(* Logix 5000 project; controller QW361 vendor 1 type 14 code 107 rev 32.11; software revision 32.00; part 18 of 20 *)

        [136].log_data[5].minminute := 7, [136].log_data[5].valid := 1, [136].log_data[6].valid := 1, [136].log_data[7].valid := 1, [136].log_data[8].valid := 1, [136].log_data[9].valid := 1, [136].log_data[10].valid := 1, [136].log_data[11].valid := 1, [136].log_data[12].valid := 1, [136].log_data[13].valid := 1, [136].log_data[14].valid := 1, [136].log_data[15].valid := 1, [136].log_data[16].valid := 1, [136].log_data[17].valid := 1, [136].log_data[18].valid := 1, [136].log_data[19].valid := 1, [136].time.Year := 2022, [136].time.Month := 5, [136].time.Day := 2, [136].time.Hour := 9, [136].time.Minute := 59, [136].time.Second := 59, [136].time.DST_ON := 1, [137].log_data[0].min := 1.0, [137].log_data[0].max := 1.0, [137].log_data[0].total := 3599.999, [137].log_data[0].time := 3599.999, [137].log_data[0].valid := 1, [137].log_data[1].max := 1.0, [137].log_data[1].total := 500.5, [137].log_data[1].time := 3599.999, [137].log_data[1].maxminute := 16, [137].log_data[1].valid := 1, [137].log_data[2].time := 3599.999, [137].log_data[2].valid := 1, [137].log_data[3].time := 3599.999, [137].log_data[3].valid := 1, [137].log_data[4].min := 0.48812497, [137].log_data[4].max := 1.0081251, [137].log_data[4].total := 2728.107, [137].log_data[4].time := 3599.999, [137].log_data[4].minminute := 25, [137].log_data[4].maxminute := 16, [137].log_data[4].valid := 1, [137].log_data[5].max := 7.1587505, [137].log_data[5].total := 3522.9197, [137].log_data[5].time := 3599.999, [137].log_data[5].maxminute := 17, [137].log_data[5].valid := 1, [137].log_data[6].valid := 1, [137].log_data[7].valid := 1, [137].log_data[8].valid := 1, [137].log_data[9].valid := 1, [137].log_data[10].valid := 1, [137].log_data[11].valid := 1, [137].log_data[12].valid := 1, [137].log_data[13].valid := 1, [137].log_data[14].valid := 1, [137].log_data[15].valid := 1, [137].log_data[16].valid := 1,
        [137].log_data[17].valid := 1, [137].log_data[18].valid := 1, [137].log_data[19].valid := 1, [137].time.Year := 2022, [137].time.Month := 5, [137].time.Day := 2, [137].time.Hour := 10, [137].time.Minute := 59, [137].time.Second := 59, [137].time.DST_ON := 1, [138].log_data[0].min := 1.0, [138].log_data[0].max := 1.0, [138].log_data[0].total := 3599.999, [138].log_data[0].time := 3599.999, [138].log_data[0].valid := 1, [138].log_data[1].time := 3599.999, [138].log_data[1].valid := 1, [138].log_data[2].max := 1.0, [138].log_data[2].total := 495.0, [138].log_data[2].time := 3599.999, [138].log_data[2].maxminute := 43, [138].log_data[2].valid := 1, [138].log_data[3].time := 3599.999, [138].log_data[3].valid := 1, [138].log_data[4].min := 0.48749998, [138].log_data[4].max := 1.0068749, [138].log_data[4].total := 3053.5842, [138].log_data[4].time := 3599.999, [138].log_data[4].minminute := 52, [138].log_data[4].maxminute := 43, [138].log_data[4].valid := 1, [138].log_data[5].max := 7.26375, [138].log_data[5].total := 3527.154, [138].log_data[5].time := 3599.999, [138].log_data[5].maxminute := 43, [138].log_data[5].valid := 1, [138].log_data[6].valid := 1, [138].log_data[7].valid := 1, [138].log_data[8].valid := 1, [138].log_data[9].valid := 1, [138].log_data[10].valid := 1, [138].log_data[11].valid := 1, [138].log_data[12].valid := 1, [138].log_data[13].valid := 1, [138].log_data[14].valid := 1, [138].log_data[15].valid := 1, [138].log_data[16].valid := 1, [138].log_data[17].valid := 1, [138].log_data[18].valid := 1, [138].log_data[19].valid := 1, [138].time.Year := 2022, [138].time.Month := 5, [138].time.Day := 2, [138].time.Hour := 11, [138].time.Minute := 59, [138].time.Second := 59, [138].time.DST_ON := 1, [139].log_data[0].min := 1.0, [139].log_data[0].max := 1.0, [139].log_data[0].total := 3599.999,
        [139].log_data[0].time := 3599.999, [139].log_data[0].valid := 1, [139].log_data[1].time := 3599.999, [139].log_data[1].valid := 1, [139].log_data[2].time := 3599.999, [139].log_data[2].valid := 1, [139].log_data[3].time := 3599.999, [139].log_data[3].valid := 1, [139].log_data[4].min := 0.56437504, [139].log_data[4].max := 0.9650001, [139].log_data[4].total := 2955.463, [139].log_data[4].time := 3599.999, [139].log_data[4].maxminute := 58, [139].log_data[4].valid := 1, [139].log_data[5].max := 0.0012500001, [139].log_data[5].total := 0.057499956, [139].log_data[5].time := 3599.999, [139].log_data[5].maxminute := 1, [139].log_data[5].valid := 1, [139].log_data[6].valid := 1, [139].log_data[7].valid := 1, [139].log_data[8].valid := 1, [139].log_data[9].valid := 1, [139].log_data[10].valid := 1, [139].log_data[11].valid := 1, [139].log_data[12].valid := 1, [139].log_data[13].valid := 1, [139].log_data[14].valid := 1, [139].log_data[15].valid := 1, [139].log_data[16].valid := 1, [139].log_data[17].valid := 1, [139].log_data[18].valid := 1, [139].log_data[19].valid := 1, [139].time.Year := 2022, [139].time.Month := 5, [139].time.Day := 2, [139].time.Hour := 12, [139].time.Minute := 59, [139].time.Second := 59, [139].time.DST_ON := 1, [140].log_data[0].min := 1.0, [140].log_data[0].max := 1.0, [140].log_data[0].total := 3600.0, [140].log_data[0].time := 3600.0, [140].log_data[0].valid := 1, [140].log_data[1].max := 1.0, [140].log_data[1].total := 501.0, [140].log_data[1].time := 3600.0, [140].log_data[1].maxminute := 9, [140].log_data[1].valid := 1, [140].log_data[2].time := 3600.0, [140].log_data[2].valid := 1, [140].log_data[3].time := 3600.0, [140].log_data[3].valid := 1, [140].log_data[4].min := 0.48749998, [140].log_data[4].max := 1.00875, [140].log_data[4].total := 2592.416, [140].log_data[4].time := 3600.0, [140].log_data[4].minminute := 18, [140].log_data[4].maxminute := 9,
        [140].log_data[4].valid := 1, [140].log_data[5].max := 7.1550007, [140].log_data[5].total := 3519.3843, [140].log_data[5].time := 3600.0, [140].log_data[5].maxminute := 10, [140].log_data[5].valid := 1, [140].log_data[6].valid := 1, [140].log_data[7].valid := 1, [140].log_data[8].valid := 1, [140].log_data[9].valid := 1, [140].log_data[10].valid := 1, [140].log_data[11].valid := 1, [140].log_data[12].valid := 1, [140].log_data[13].valid := 1, [140].log_data[14].valid := 1, [140].log_data[15].valid := 1, [140].log_data[16].valid := 1, [140].log_data[17].valid := 1, [140].log_data[18].valid := 1, [140].log_data[19].valid := 1, [140].time.Year := 2022, [140].time.Month := 5, [140].time.Day := 2, [140].time.Hour := 13, [140].time.Minute := 59, [140].time.Second := 59, [140].time.DST_ON := 1, [141].log_data[0].min := 1.0, [141].log_data[0].max := 1.0, [141].log_data[0].total := 3600.001, [141].log_data[0].time := 3600.001, [141].log_data[0].valid := 1, [141].log_data[1].time := 3600.001, [141].log_data[1].valid := 1, [141].log_data[2].time := 3600.001, [141].log_data[2].valid := 1, [141].log_data[3].time := 3600.001, [141].log_data[3].valid := 1, [141].log_data[4].min := 0.77937496, [141].log_data[4].max := 0.94875, [141].log_data[4].total := 3176.0435, [141].log_data[4].time := 3600.001, [141].log_data[4].maxminute := 56, [141].log_data[4].valid := 1, [141].log_data[5].max := 0.0012500001, [141].log_data[5].total := 0.14781292, [141].log_data[5].time := 3600.001, [141].log_data[5].valid := 1, [141].log_data[6].valid := 1, [141].log_data[7].valid := 1, [141].log_data[8].valid := 1, [141].log_data[9].valid := 1, [141].log_data[10].valid := 1, [141].log_data[11].valid := 1, [141].log_data[12].valid := 1, [141].log_data[13].valid := 1, [141].log_data[14].valid := 1, [141].log_data[15].valid := 1, [141].log_data[16].valid := 1, [141].log_data[17].valid := 1,
        [141].log_data[18].valid := 1, [141].log_data[19].valid := 1, [141].time.Year := 2022, [141].time.Month := 5, [141].time.Day := 2, [141].time.Hour := 14, [141].time.Minute := 59, [141].time.Second := 59, [141].time.DST_ON := 1, [142].log_data[0].min := 1.0, [142].log_data[0].max := 1.0, [142].log_data[0].total := 3600.0, [142].log_data[0].time := 3600.0, [142].log_data[0].valid := 1, [142].log_data[1].time := 3600.0, [142].log_data[1].valid := 1, [142].log_data[2].max := 1.0, [142].log_data[2].total := 480.0, [142].log_data[2].time := 3600.0, [142].log_data[2].maxminute := 26, [142].log_data[2].valid := 1, [142].log_data[3].time := 3600.0, [142].log_data[3].valid := 1, [142].log_data[4].min := 0.48749998, [142].log_data[4].max := 1.00625, [142].log_data[4].total := 2781.7415, [142].log_data[4].time := 3600.0, [142].log_data[4].minminute := 34, [142].log_data[4].maxminute := 26, [142].log_data[4].valid := 1, [142].log_data[5].max := 7.3075004, [142].log_data[5].total := 3444.1716, [142].log_data[5].time := 3600.0, [142].log_data[5].maxminute := 27, [142].log_data[5].valid := 1, [142].log_data[6].valid := 1, [142].log_data[7].valid := 1, [142].log_data[8].valid := 1, [142].log_data[9].valid := 1, [142].log_data[10].valid := 1, [142].log_data[11].valid := 1, [142].log_data[12].valid := 1, [142].log_data[13].valid := 1, [142].log_data[14].valid := 1, [142].log_data[15].valid := 1, [142].log_data[16].valid := 1, [142].log_data[17].valid := 1, [142].log_data[18].valid := 1, [142].log_data[19].valid := 1, [142].time.Year := 2022, [142].time.Month := 5, [142].time.Day := 2, [142].time.Hour := 15, [142].time.Minute := 59, [142].time.Second := 59, [142].time.DST_ON := 1, [143].log_data[0].min := 1.0, [143].log_data[0].max := 1.0, [143].log_data[0].total := 3599.999, [143].log_data[0].time := 3599.999,
        [143].log_data[0].valid := 1, [143].log_data[1].time := 3599.999, [143].log_data[1].valid := 1, [143].log_data[2].time := 3599.999, [143].log_data[2].valid := 1, [143].log_data[3].time := 3599.999, [143].log_data[3].valid := 1, [143].log_data[4].min := 0.64125, [143].log_data[4].max := 0.97937495, [143].log_data[4].total := 2973.9944, [143].log_data[4].time := 3599.999, [143].log_data[4].maxminute := 57, [143].log_data[4].valid := 1, [143].log_data[5].time := 3599.999, [143].log_data[5].valid := 1, [143].log_data[6].valid := 1, [143].log_data[7].valid := 1, [143].log_data[8].valid := 1, [143].log_data[9].valid := 1, [143].log_data[10].valid := 1, [143].log_data[11].valid := 1, [143].log_data[12].valid := 1, [143].log_data[13].valid := 1, [143].log_data[14].valid := 1, [143].log_data[15].valid := 1, [143].log_data[16].valid := 1, [143].log_data[17].valid := 1, [143].log_data[18].valid := 1, [143].log_data[19].valid := 1, [143].time.Year := 2022, [143].time.Month := 5, [143].time.Day := 2, [143].time.Hour := 16, [143].time.Minute := 59, [143].time.Second := 59, [143].time.DST_ON := 1, [144].log_data[0].min := 1.0, [144].log_data[0].max := 1.0, [144].log_data[0].total := 3600.0, [144].log_data[0].time := 3600.0, [144].log_data[0].valid := 1, [144].log_data[1].max := 1.0, [144].log_data[1].total := 497.5, [144].log_data[1].time := 3600.0, [144].log_data[1].maxminute := 6, [144].log_data[1].valid := 1, [144].log_data[2].time := 3600.0, [144].log_data[2].valid := 1, [144].log_data[3].time := 3600.0, [144].log_data[3].valid := 1, [144].log_data[4].min := 0.48749998, [144].log_data[4].max := 1.00875, [144].log_data[4].total := 2580.9526, [144].log_data[4].time := 3600.0, [144].log_data[4].minminute := 15, [144].log_data[4].maxminute := 6, [144].log_data[4].valid := 1, [144].log_data[5].max := 7.1587505, [144].log_data[5].total := 3498.0137, [144].log_data[5].time := 3600.0,
        [144].log_data[5].maxminute := 8, [144].log_data[5].valid := 1, [144].log_data[6].valid := 1, [144].log_data[7].valid := 1, [144].log_data[8].valid := 1, [144].log_data[9].valid := 1, [144].log_data[10].valid := 1, [144].log_data[11].valid := 1, [144].log_data[12].valid := 1, [144].log_data[13].valid := 1, [144].log_data[14].valid := 1, [144].log_data[15].valid := 1, [144].log_data[16].valid := 1, [144].log_data[17].valid := 1, [144].log_data[18].valid := 1, [144].log_data[19].valid := 1, [144].time.Year := 2022, [144].time.Month := 5, [144].time.Day := 2, [144].time.Hour := 17, [144].time.Minute := 59, [144].time.Second := 59, [144].time.DST_ON := 1, [145].log_data[0].min := 1.0, [145].log_data[0].max := 1.0, [145].log_data[0].total := 3600.0, [145].log_data[0].time := 3600.0, [145].log_data[0].valid := 1, [145].log_data[1].time := 3600.0, [145].log_data[1].valid := 1, [145].log_data[2].max := 1.0, [145].log_data[2].total := 489.5, [145].log_data[2].time := 3600.0, [145].log_data[2].maxminute := 45, [145].log_data[2].valid := 1, [145].log_data[3].time := 3600.0, [145].log_data[3].valid := 1, [145].log_data[4].min := 0.48749998, [145].log_data[4].max := 1.00875, [145].log_data[4].total := 3124.9949, [145].log_data[4].time := 3600.0, [145].log_data[4].minminute := 53, [145].log_data[4].maxminute := 45, [145].log_data[4].valid := 1, [145].log_data[5].max := 7.2675, [145].log_data[5].total := 3485.3735, [145].log_data[5].time := 3600.0, [145].log_data[5].maxminute := 46, [145].log_data[5].valid := 1, [145].log_data[6].valid := 1, [145].log_data[7].valid := 1, [145].log_data[8].valid := 1, [145].log_data[9].valid := 1, [145].log_data[10].valid := 1, [145].log_data[11].valid := 1, [145].log_data[12].valid := 1, [145].log_data[13].valid := 1, [145].log_data[14].valid := 1, [145].log_data[15].valid := 1, [145].log_data[16].valid := 1,
        [145].log_data[17].valid := 1, [145].log_data[18].valid := 1, [145].log_data[19].valid := 1, [145].time.Year := 2022, [145].time.Month := 5, [145].time.Day := 2, [145].time.Hour := 18, [145].time.Minute := 59, [145].time.Second := 59, [145].time.DST_ON := 1, [146].log_data[0].min := 1.0, [146].log_data[0].max := 1.0, [146].log_data[0].total := 3600.0, [146].log_data[0].time := 3600.0, [146].log_data[0].valid := 1, [146].log_data[1].time := 3600.0, [146].log_data[1].valid := 1, [146].log_data[2].time := 3600.0, [146].log_data[2].valid := 1, [146].log_data[3].time := 3600.0, [146].log_data[3].valid := 1, [146].log_data[4].min := 0.53374994, [146].log_data[4].max := 0.933125, [146].log_data[4].total := 2734.3828, [146].log_data[4].time := 3600.0, [146].log_data[4].maxminute := 58, [146].log_data[4].valid := 1, [146].log_data[5].time := 3600.0, [146].log_data[5].valid := 1, [146].log_data[6].valid := 1, [146].log_data[7].valid := 1, [146].log_data[8].valid := 1, [146].log_data[9].valid := 1, [146].log_data[10].valid := 1, [146].log_data[11].valid := 1, [146].log_data[12].valid := 1, [146].log_data[13].valid := 1, [146].log_data[14].valid := 1, [146].log_data[15].valid := 1, [146].log_data[16].valid := 1, [146].log_data[17].valid := 1, [146].log_data[18].valid := 1, [146].log_data[19].valid := 1, [146].time.Year := 2022, [146].time.Month := 5, [146].time.Day := 2, [146].time.Hour := 19, [146].time.Minute := 59, [146].time.Second := 59, [146].time.DST_ON := 1, [147].log_data[0].min := 1.0, [147].log_data[0].max := 1.0, [147].log_data[0].total := 3600.0, [147].log_data[0].time := 3600.0, [147].log_data[0].valid := 1, [147].log_data[1].max := 1.0, [147].log_data[1].total := 512.0, [147].log_data[1].time := 3600.0, [147].log_data[1].maxminute := 17, [147].log_data[1].valid := 1,
        [147].log_data[2].time := 3600.0, [147].log_data[2].valid := 1, [147].log_data[3].time := 3600.0, [147].log_data[3].valid := 1, [147].log_data[4].min := 0.48749998, [147].log_data[4].max := 1.00875, [147].log_data[4].total := 2863.854, [147].log_data[4].time := 3600.0, [147].log_data[4].minminute := 26, [147].log_data[4].maxminute := 18, [147].log_data[4].valid := 1, [147].log_data[5].max := 7.1587505, [147].log_data[5].total := 3600.5417, [147].log_data[5].time := 3600.0, [147].log_data[5].maxminute := 18, [147].log_data[5].valid := 1, [147].log_data[6].valid := 1, [147].log_data[7].valid := 1, [147].log_data[8].valid := 1, [147].log_data[9].valid := 1, [147].log_data[10].valid := 1, [147].log_data[11].valid := 1, [147].log_data[12].valid := 1, [147].log_data[13].valid := 1, [147].log_data[14].valid := 1, [147].log_data[15].valid := 1, [147].log_data[16].valid := 1, [147].log_data[17].valid := 1, [147].log_data[18].valid := 1, [147].log_data[19].valid := 1, [147].time.Year := 2022, [147].time.Month := 5, [147].time.Day := 2, [147].time.Hour := 20, [147].time.Minute := 59, [147].time.Second := 59, [147].time.DST_ON := 1, [148].log_data[0].min := 1.0, [148].log_data[0].max := 1.0, [148].log_data[0].total := 3600.0, [148].log_data[0].time := 3600.0, [148].log_data[0].valid := 1, [148].log_data[1].time := 3600.0, [148].log_data[1].valid := 1, [148].log_data[2].max := 1.0, [148].log_data[2].total := 498.0, [148].log_data[2].time := 3600.0, [148].log_data[2].maxminute := 20, [148].log_data[2].valid := 1, [148].log_data[3].time := 3600.0, [148].log_data[3].valid := 1, [148].log_data[4].min := 0.48749998, [148].log_data[4].max := 1.00875, [148].log_data[4].total := 2776.5615, [148].log_data[4].time := 3600.0, [148].log_data[4].minminute := 28, [148].log_data[4].maxminute := 20, [148].log_data[4].valid := 1, [148].log_data[5].max := 7.2425003, [148].log_data[5].total := 3543.449,
        [148].log_data[5].time := 3600.0, [148].log_data[5].maxminute := 21, [148].log_data[5].valid := 1, [148].log_data[6].valid := 1, [148].log_data[7].valid := 1, [148].log_data[8].valid := 1, [148].log_data[9].valid := 1, [148].log_data[10].valid := 1, [148].log_data[11].valid := 1, [148].log_data[12].valid := 1, [148].log_data[13].valid := 1, [148].log_data[14].valid := 1, [148].log_data[15].valid := 1, [148].log_data[16].valid := 1, [148].log_data[17].valid := 1, [148].log_data[18].valid := 1, [148].log_data[19].valid := 1, [148].time.Year := 2022, [148].time.Month := 5, [148].time.Day := 2, [148].time.Hour := 21, [148].time.Minute := 59, [148].time.Second := 59, [148].time.DST_ON := 1, [149].log_data[0].min := 1.0, [149].log_data[0].max := 1.0, [149].log_data[0].total := 3600.0, [149].log_data[0].time := 3600.0, [149].log_data[0].valid := 1, [149].log_data[1].max := 1.0, [149].log_data[1].total := 509.5, [149].log_data[1].time := 3600.0, [149].log_data[1].maxminute := 25, [149].log_data[1].valid := 1, [149].log_data[2].time := 3600.0, [149].log_data[2].valid := 1, [149].log_data[3].time := 3600.0, [149].log_data[3].valid := 1, [149].log_data[4].min := 0.48749998, [149].log_data[4].max := 1.00875, [149].log_data[4].total := 2806.5916, [149].log_data[4].time := 3600.0, [149].log_data[4].minminute := 34, [149].log_data[4].maxminute := 25, [149].log_data[4].valid := 1, [149].log_data[5].max := 7.1662498, [149].log_data[5].total := 3591.45, [149].log_data[5].time := 3600.0, [149].log_data[5].maxminute := 26, [149].log_data[5].valid := 1, [149].log_data[6].valid := 1, [149].log_data[7].valid := 1, [149].log_data[8].valid := 1, [149].log_data[9].valid := 1, [149].log_data[10].valid := 1, [149].log_data[11].valid := 1, [149].log_data[12].valid := 1, [149].log_data[13].valid := 1, [149].log_data[14].valid := 1, [149].log_data[15].valid := 1,
        [149].log_data[16].valid := 1, [149].log_data[17].valid := 1, [149].log_data[18].valid := 1, [149].log_data[19].valid := 1, [149].time.Year := 2022, [149].time.Month := 5, [149].time.Day := 2, [149].time.Hour := 22, [149].time.Minute := 59, [149].time.Second := 59, [149].time.DST_ON := 1, [150].log_data[0].min := 1.0, [150].log_data[0].max := 1.0, [150].log_data[0].total := 3600.0, [150].log_data[0].time := 3600.0, [150].log_data[0].valid := 1, [150].log_data[1].time := 3600.0, [150].log_data[1].valid := 1, [150].log_data[2].max := 1.0, [150].log_data[2].total := 488.5, [150].log_data[2].time := 3600.0, [150].log_data[2].maxminute := 42, [150].log_data[2].valid := 1, [150].log_data[3].time := 3600.0, [150].log_data[3].valid := 1, [150].log_data[4].min := 0.48749998, [150].log_data[4].max := 1.0068749, [150].log_data[4].total := 3012.5884, [150].log_data[4].time := 3600.0, [150].log_data[4].minminute := 51, [150].log_data[4].maxminute := 42, [150].log_data[4].valid := 1, [150].log_data[5].max := 7.2337503, [150].log_data[5].total := 3473.9883, [150].log_data[5].time := 3600.0, [150].log_data[5].maxminute := 43, [150].log_data[5].valid := 1, [150].log_data[6].valid := 1, [150].log_data[7].valid := 1, [150].log_data[8].valid := 1, [150].log_data[9].valid := 1, [150].log_data[10].valid := 1, [150].log_data[11].valid := 1, [150].log_data[12].valid := 1, [150].log_data[13].valid := 1, [150].log_data[14].valid := 1, [150].log_data[15].valid := 1, [150].log_data[16].valid := 1, [150].log_data[17].valid := 1, [150].log_data[18].valid := 1, [150].log_data[19].valid := 1, [150].time.Year := 2022, [150].time.Month := 5, [150].time.Day := 2, [150].time.Hour := 23, [150].time.Minute := 59, [150].time.Second := 59, [150].time.DST_ON := 1, [151].log_data[0].min := 1.0, [151].log_data[0].max := 1.0,
        [151].log_data[0].total := 3599.999, [151].log_data[0].time := 3599.999, [151].log_data[0].valid := 1, [151].log_data[1].time := 3599.999, [151].log_data[1].valid := 1, [151].log_data[2].time := 3599.999, [151].log_data[2].valid := 1, [151].log_data[3].time := 3599.999, [151].log_data[3].valid := 1, [151].log_data[4].min := 0.549375, [151].log_data[4].max := 0.91875005, [151].log_data[4].total := 2695.1277, [151].log_data[4].time := 3599.999, [151].log_data[4].maxminute := 57, [151].log_data[4].valid := 1, [151].log_data[5].max := 0.0012500001, [151].log_data[5].total := 0.15468808, [151].log_data[5].time := 3599.999, [151].log_data[5].valid := 1, [151].log_data[6].valid := 1, [151].log_data[7].valid := 1, [151].log_data[8].valid := 1, [151].log_data[9].valid := 1, [151].log_data[10].valid := 1, [151].log_data[11].valid := 1, [151].log_data[12].valid := 1, [151].log_data[13].valid := 1, [151].log_data[14].valid := 1, [151].log_data[15].valid := 1, [151].log_data[16].valid := 1, [151].log_data[17].valid := 1, [151].log_data[18].valid := 1, [151].log_data[19].valid := 1, [151].time.Year := 2022, [151].time.Month := 5, [151].time.Day := 3, [151].time.Minute := 59, [151].time.Second := 59, [151].time.DST_ON := 1, [152].log_data[0].min := 1.0, [152].log_data[0].max := 1.0, [152].log_data[0].total := 3600.0, [152].log_data[0].time := 3600.0, [152].log_data[0].valid := 1, [152].log_data[1].max := 1.0, [152].log_data[1].total := 480.0, [152].log_data[1].time := 3600.0, [152].log_data[1].maxminute := 32, [152].log_data[1].valid := 1, [152].log_data[2].time := 3600.0, [152].log_data[2].valid := 1, [152].log_data[3].time := 3600.0, [152].log_data[3].valid := 1, [152].log_data[4].min := 0.48812497, [152].log_data[4].max := 1.00625, [152].log_data[4].total := 2904.3708, [152].log_data[4].time := 3600.0, [152].log_data[4].minminute := 40, [152].log_data[4].maxminute := 32, [152].log_data[4].valid := 1,
        [152].log_data[5].max := 7.26375, [152].log_data[5].total := 3427.8037, [152].log_data[5].time := 3600.0, [152].log_data[5].maxminute := 34, [152].log_data[5].valid := 1, [152].log_data[6].valid := 1, [152].log_data[7].valid := 1, [152].log_data[8].valid := 1, [152].log_data[9].valid := 1, [152].log_data[10].valid := 1, [152].log_data[11].valid := 1, [152].log_data[12].valid := 1, [152].log_data[13].valid := 1, [152].log_data[14].valid := 1, [152].log_data[15].valid := 1, [152].log_data[16].valid := 1, [152].log_data[17].valid := 1, [152].log_data[18].valid := 1, [152].log_data[19].valid := 1, [152].time.Year := 2022, [152].time.Month := 5, [152].time.Day := 3, [152].time.Hour := 1, [152].time.Minute := 59, [152].time.Second := 59, [152].time.DST_ON := 1, [153].log_data[0].min := 1.0, [153].log_data[0].max := 1.0, [153].log_data[0].total := 3599.999, [153].log_data[0].time := 3599.999, [153].log_data[0].valid := 1, [153].log_data[1].time := 3599.999, [153].log_data[1].valid := 1, [153].log_data[2].time := 3599.999, [153].log_data[2].valid := 1, [153].log_data[3].time := 3599.999, [153].log_data[3].valid := 1, [153].log_data[4].min := 0.610625, [153].log_data[4].max := 0.841875, [153].log_data[4].total := 2696.8096, [153].log_data[4].time := 3599.999, [153].log_data[4].maxminute := 56, [153].log_data[4].valid := 1, [153].log_data[5].max := 0.0012500001, [153].log_data[5].total := 0.11062366, [153].log_data[5].time := 3599.999, [153].log_data[5].valid := 1, [153].log_data[6].valid := 1, [153].log_data[7].valid := 1, [153].log_data[8].valid := 1, [153].log_data[9].valid := 1, [153].log_data[10].valid := 1, [153].log_data[11].valid := 1, [153].log_data[12].valid := 1, [153].log_data[13].valid := 1, [153].log_data[14].valid := 1, [153].log_data[15].valid := 1, [153].log_data[16].valid := 1, [153].log_data[17].valid := 1, [153].log_data[18].valid := 1,
        [153].log_data[19].valid := 1, [153].time.Year := 2022, [153].time.Month := 5, [153].time.Day := 3, [153].time.Hour := 2, [153].time.Minute := 59, [153].time.Second := 59, [153].time.DST_ON := 1, [154].log_data[0].min := 1.0, [154].log_data[0].max := 1.0, [154].log_data[0].total := 3600.0, [154].log_data[0].time := 3600.0, [154].log_data[0].valid := 1, [154].log_data[1].time := 3600.0, [154].log_data[1].valid := 1, [154].log_data[2].time := 3600.0, [154].log_data[2].valid := 1, [154].log_data[3].time := 3600.0, [154].log_data[3].valid := 1, [154].log_data[4].min := 0.84124994, [154].log_data[4].max := 0.91875005, [154].log_data[4].total := 3198.6758, [154].log_data[4].time := 3600.0, [154].log_data[4].maxminute := 49, [154].log_data[4].valid := 1, [154].log_data[5].max := 0.0012500001, [154].log_data[5].total := 0.04156247, [154].log_data[5].time := 3600.0, [154].log_data[5].maxminute := 1, [154].log_data[5].valid := 1, [154].log_data[6].valid := 1, [154].log_data[7].valid := 1, [154].log_data[8].valid := 1, [154].log_data[9].valid := 1, [154].log_data[10].valid := 1, [154].log_data[11].valid := 1, [154].log_data[12].valid := 1, [154].log_data[13].valid := 1, [154].log_data[14].valid := 1, [154].log_data[15].valid := 1, [154].log_data[16].valid := 1, [154].log_data[17].valid := 1, [154].log_data[18].valid := 1, [154].log_data[19].valid := 1, [154].time.Year := 2022, [154].time.Month := 5, [154].time.Day := 3, [154].time.Hour := 3, [154].time.Minute := 59, [154].time.Second := 59, [154].time.DST_ON := 1, [155].log_data[0].min := 1.0, [155].log_data[0].max := 1.0, [155].log_data[0].total := 3600.0, [155].log_data[0].time := 3600.0, [155].log_data[0].valid := 1, [155].log_data[1].time := 3600.0, [155].log_data[1].valid := 1, [155].log_data[2].time := 3600.0, [155].log_data[2].valid := 1,
        [155].log_data[3].time := 3600.0, [155].log_data[3].valid := 1, [155].log_data[4].min := 0.918125, [155].log_data[4].max := 0.9650001, [155].log_data[4].total := 3389.3665, [155].log_data[4].time := 3600.0, [155].log_data[4].maxminute := 54, [155].log_data[4].valid := 1, [155].log_data[5].max := 0.0012500001, [155].log_data[5].total := 0.056874957, [155].log_data[5].time := 3600.0, [155].log_data[5].valid := 1, [155].log_data[6].valid := 1, [155].log_data[7].valid := 1, [155].log_data[8].valid := 1, [155].log_data[9].valid := 1, [155].log_data[10].valid := 1, [155].log_data[11].valid := 1, [155].log_data[12].valid := 1, [155].log_data[13].valid := 1, [155].log_data[14].valid := 1, [155].log_data[15].valid := 1, [155].log_data[16].valid := 1, [155].log_data[17].valid := 1, [155].log_data[18].valid := 1, [155].log_data[19].valid := 1, [155].time.Year := 2022, [155].time.Month := 5, [155].time.Day := 3, [155].time.Hour := 4, [155].time.Minute := 59, [155].time.Second := 59, [155].time.DST_ON := 1, [156].log_data[0].min := 1.0, [156].log_data[0].max := 1.0, [156].log_data[0].total := 3600.001, [156].log_data[0].time := 3600.001, [156].log_data[0].valid := 1, [156].log_data[1].time := 3600.001, [156].log_data[1].valid := 1, [156].log_data[2].max := 1.0, [156].log_data[2].total := 478.0, [156].log_data[2].time := 3600.001, [156].log_data[2].maxminute := 20, [156].log_data[2].valid := 1, [156].log_data[3].time := 3600.001, [156].log_data[3].valid := 1, [156].log_data[4].min := 0.48812497, [156].log_data[4].max := 1.0068749, [156].log_data[4].total := 2638.017, [156].log_data[4].time := 3600.001, [156].log_data[4].minminute := 28, [156].log_data[4].maxminute := 20, [156].log_data[4].valid := 1, [156].log_data[5].max := 7.2512507, [156].log_data[5].total := 3407.9675, [156].log_data[5].time := 3600.001, [156].log_data[5].maxminute := 22, [156].log_data[5].valid := 1, [156].log_data[6].valid := 1,
        [156].log_data[7].valid := 1, [156].log_data[8].valid := 1, [156].log_data[9].valid := 1, [156].log_data[10].valid := 1, [156].log_data[11].valid := 1, [156].log_data[12].valid := 1, [156].log_data[13].valid := 1, [156].log_data[14].valid := 1, [156].log_data[15].valid := 1, [156].log_data[16].valid := 1, [156].log_data[17].valid := 1, [156].log_data[18].valid := 1, [156].log_data[19].valid := 1, [156].time.Year := 2022, [156].time.Month := 5, [156].time.Day := 3, [156].time.Hour := 5, [156].time.Minute := 59, [156].time.Second := 59, [156].time.DST_ON := 1, [157].log_data[0].min := 1.0, [157].log_data[0].max := 1.0, [157].log_data[0].total := 3600.0, [157].log_data[0].time := 3600.0, [157].log_data[0].valid := 1, [157].log_data[1].time := 3600.0, [157].log_data[1].valid := 1, [157].log_data[2].time := 3600.0, [157].log_data[2].valid := 1, [157].log_data[3].time := 3600.0, [157].log_data[3].valid := 1, [157].log_data[4].min := 0.625625, [157].log_data[4].max := 0.76437503, [157].log_data[4].total := 2547.3604, [157].log_data[4].time := 3600.0, [157].log_data[4].maxminute := 54, [157].log_data[4].valid := 1, [157].log_data[5].max := 0.0012500001, [157].log_data[5].total := 0.13343759, [157].log_data[5].time := 3600.0, [157].log_data[5].valid := 1, [157].log_data[6].valid := 1, [157].log_data[7].valid := 1, [157].log_data[8].valid := 1, [157].log_data[9].valid := 1, [157].log_data[10].valid := 1, [157].log_data[11].valid := 1, [157].log_data[12].valid := 1, [157].log_data[13].valid := 1, [157].log_data[14].valid := 1, [157].log_data[15].valid := 1, [157].log_data[16].valid := 1, [157].log_data[17].valid := 1, [157].log_data[18].valid := 1, [157].log_data[19].valid := 1, [157].time.Year := 2022, [157].time.Month := 5, [157].time.Day := 3, [157].time.Hour := 6, [157].time.Minute := 59,
        [157].time.Second := 59, [157].time.DST_ON := 1, [158].log_data[0].min := 1.0, [158].log_data[0].max := 1.0, [158].log_data[0].total := 3599.999, [158].log_data[0].time := 3599.999, [158].log_data[0].valid := 1, [158].log_data[1].time := 3599.999, [158].log_data[1].valid := 1, [158].log_data[2].time := 3599.999, [158].log_data[2].valid := 1, [158].log_data[3].time := 3599.999, [158].log_data[3].valid := 1, [158].log_data[4].min := 0.76375, [158].log_data[4].max := 0.9024999, [158].log_data[4].total := 2931.7944, [158].log_data[4].time := 3599.999, [158].log_data[4].maxminute := 58, [158].log_data[4].valid := 1, [158].log_data[5].max := 0.0012500001, [158].log_data[5].total := 0.1296875, [158].log_data[5].time := 3599.999, [158].log_data[5].valid := 1, [158].log_data[6].valid := 1, [158].log_data[7].valid := 1, [158].log_data[8].valid := 1, [158].log_data[9].valid := 1, [158].log_data[10].valid := 1, [158].log_data[11].valid := 1, [158].log_data[12].valid := 1, [158].log_data[13].valid := 1, [158].log_data[14].valid := 1, [158].log_data[15].valid := 1, [158].log_data[16].valid := 1, [158].log_data[17].valid := 1, [158].log_data[18].valid := 1, [158].log_data[19].valid := 1, [158].time.Year := 2022, [158].time.Month := 5, [158].time.Day := 3, [158].time.Hour := 7, [158].time.Minute := 59, [158].time.Second := 59, [158].time.DST_ON := 1, [159].log_data[0].min := 1.0, [159].log_data[0].max := 1.0, [159].log_data[0].total := 3600.0, [159].log_data[0].time := 3600.0, [159].log_data[0].valid := 1, [159].log_data[1].max := 1.0, [159].log_data[1].total := 629.5, [159].log_data[1].time := 3600.0, [159].log_data[1].maxminute := 28, [159].log_data[1].valid := 1, [159].log_data[2].time := 3600.0, [159].log_data[2].valid := 1, [159].log_data[3].time := 3600.0, [159].log_data[3].valid := 1, [159].log_data[4].min := 0.48812497, [159].log_data[4].max := 1.00625,
        [159].log_data[4].total := 2832.5337, [159].log_data[4].time := 3600.0, [159].log_data[4].minminute := 36, [159].log_data[4].maxminute := 28, [159].log_data[4].valid := 1, [159].log_data[5].max := 7.1699996, [159].log_data[5].total := 4413.0254, [159].log_data[5].time := 3600.0, [159].log_data[5].maxminute := 28, [159].log_data[5].valid := 1, [159].log_data[6].valid := 1, [159].log_data[7].valid := 1, [159].log_data[8].valid := 1, [159].log_data[9].valid := 1, [159].log_data[10].valid := 1, [159].log_data[11].valid := 1, [159].log_data[12].valid := 1, [159].log_data[13].valid := 1, [159].log_data[14].valid := 1, [159].log_data[15].valid := 1, [159].log_data[16].valid := 1, [159].log_data[17].valid := 1, [159].log_data[18].valid := 1, [159].log_data[19].valid := 1, [159].time.Year := 2022, [159].time.Month := 5, [159].time.Day := 3, [159].time.Hour := 8, [159].time.Minute := 59, [159].time.Second := 59, [159].time.DST_ON := 1, [160].log_data[0].min := 1.0, [160].log_data[0].max := 1.0, [160].log_data[0].total := 3600.0, [160].log_data[0].time := 3600.0, [160].log_data[0].valid := 1, [160].log_data[1].time := 3600.0, [160].log_data[1].valid := 1, [160].log_data[2].time := 3600.0, [160].log_data[2].valid := 1, [160].log_data[3].time := 3600.0, [160].log_data[3].valid := 1, [160].log_data[4].min := 0.55, [160].log_data[4].max := 0.9650001, [160].log_data[4].total := 2898.0752, [160].log_data[4].time := 3600.0, [160].log_data[4].maxminute := 55, [160].log_data[4].valid := 1, [160].log_data[5].max := 0.0012500001, [160].log_data[5].total := 0.25625288, [160].log_data[5].time := 3600.0, [160].log_data[5].valid := 1, [160].log_data[6].valid := 1, [160].log_data[7].valid := 1, [160].log_data[8].valid := 1, [160].log_data[9].valid := 1, [160].log_data[10].valid := 1, [160].log_data[11].valid := 1, [160].log_data[12].valid := 1, [160].log_data[13].valid := 1,
        [160].log_data[14].valid := 1, [160].log_data[15].valid := 1, [160].log_data[16].valid := 1, [160].log_data[17].valid := 1, [160].log_data[18].valid := 1, [160].log_data[19].valid := 1, [160].time.Year := 2022, [160].time.Month := 5, [160].time.Day := 3, [160].time.Hour := 9, [160].time.Minute := 59, [160].time.Second := 59, [160].time.DST_ON := 1, [161].log_data[0].min := 1.0, [161].log_data[0].max := 1.0, [161].log_data[0].total := 3600.0, [161].log_data[0].time := 3600.0, [161].log_data[0].valid := 1, [161].log_data[1].time := 3600.0, [161].log_data[1].valid := 1, [161].log_data[2].max := 1.0, [161].log_data[2].total := 483.5, [161].log_data[2].time := 3600.0, [161].log_data[2].maxminute := 13, [161].log_data[2].valid := 1, [161].log_data[3].time := 3600.0, [161].log_data[3].valid := 1, [161].log_data[4].min := 0.48749998, [161].log_data[4].max := 1.00625, [161].log_data[4].total := 2543.284, [161].log_data[4].time := 3600.0, [161].log_data[4].minminute := 21, [161].log_data[4].maxminute := 13, [161].log_data[4].valid := 1, [161].log_data[5].max := 7.241251, [161].log_data[5].total := 3439.7163, [161].log_data[5].time := 3600.0, [161].log_data[5].maxminute := 15, [161].log_data[5].valid := 1, [161].log_data[6].valid := 1, [161].log_data[7].valid := 1, [161].log_data[8].valid := 1, [161].log_data[9].valid := 1, [161].log_data[10].valid := 1, [161].log_data[11].valid := 1, [161].log_data[12].valid := 1, [161].log_data[13].valid := 1, [161].log_data[14].valid := 1, [161].log_data[15].valid := 1, [161].log_data[16].valid := 1, [161].log_data[17].valid := 1, [161].log_data[18].valid := 1, [161].log_data[19].valid := 1, [161].time.Year := 2022, [161].time.Month := 5, [161].time.Day := 3, [161].time.Hour := 10, [161].time.Minute := 59, [161].time.Second := 59, [161].time.DST_ON := 1,
        [162].log_data[0].min := 1.0, [162].log_data[0].max := 1.0, [162].log_data[0].total := 3600.0, [162].log_data[0].time := 3600.0, [162].log_data[0].valid := 1, [162].log_data[1].time := 3600.0, [162].log_data[1].valid := 1, [162].log_data[2].time := 3600.0, [162].log_data[2].valid := 1, [162].log_data[3].time := 3600.0, [162].log_data[3].valid := 1, [162].log_data[4].min := 0.703125, [162].log_data[4].max := 0.994375, [162].log_data[4].total := 3179.3467, [162].log_data[4].time := 3600.0, [162].log_data[4].maxminute := 55, [162].log_data[4].valid := 1, [162].log_data[5].time := 3600.0, [162].log_data[5].valid := 1, [162].log_data[6].valid := 1, [162].log_data[7].valid := 1, [162].log_data[8].valid := 1, [162].log_data[9].valid := 1, [162].log_data[10].valid := 1, [162].log_data[11].valid := 1, [162].log_data[12].valid := 1, [162].log_data[13].valid := 1, [162].log_data[14].valid := 1, [162].log_data[15].valid := 1, [162].log_data[16].valid := 1, [162].log_data[17].valid := 1, [162].log_data[18].valid := 1, [162].log_data[19].valid := 1, [162].time.Year := 2022, [162].time.Month := 5, [162].time.Day := 3, [162].time.Hour := 11, [162].time.Minute := 59, [162].time.Second := 59, [162].time.DST_ON := 1, [163].log_data[0].min := 1.0, [163].log_data[0].max := 1.0, [163].log_data[0].total := 3600.0, [163].log_data[0].time := 3600.0, [163].log_data[0].valid := 1, [163].log_data[1].max := 1.0, [163].log_data[1].total := 634.75, [163].log_data[1].time := 3600.0, [163].log_data[1].maxminute := 1, [163].log_data[1].valid := 1, [163].log_data[2].max := 1.0, [163].log_data[2].total := 130.5, [163].log_data[2].time := 3600.0, [163].log_data[2].maxminute := 49, [163].log_data[2].valid := 1, [163].log_data[3].time := 3600.0, [163].log_data[3].valid := 1, [163].log_data[4].min := 0.48749998, [163].log_data[4].max := 1.00625, [163].log_data[4].total := 2403.324,
        [163].log_data[4].time := 3600.0, [163].log_data[4].minminute := 9, [163].log_data[4].maxminute := 1, [163].log_data[4].valid := 1, [163].log_data[5].max := 8.66, [163].log_data[5].total := 4654.9297, [163].log_data[5].time := 3600.0, [163].log_data[5].maxminute := 50, [163].log_data[5].valid := 1, [163].log_data[6].valid := 1, [163].log_data[7].valid := 1, [163].log_data[8].valid := 1, [163].log_data[9].valid := 1, [163].log_data[10].valid := 1, [163].log_data[11].valid := 1, [163].log_data[12].valid := 1, [163].log_data[13].valid := 1, [163].log_data[14].valid := 1, [163].log_data[15].valid := 1, [163].log_data[16].valid := 1, [163].log_data[17].valid := 1, [163].log_data[18].valid := 1, [163].log_data[19].valid := 1, [163].time.Year := 2022, [163].time.Month := 5, [163].time.Day := 3, [163].time.Hour := 12, [163].time.Minute := 59, [163].time.Second := 59, [163].time.DST_ON := 1, [164].log_data[0].min := 1.0, [164].log_data[0].max := 1.0, [164].log_data[0].total := 3600.0, [164].log_data[0].time := 3600.0, [164].log_data[0].valid := 1, [164].log_data[1].time := 3600.0, [164].log_data[1].valid := 1, [164].log_data[2].time := 3600.0, [164].log_data[2].valid := 1, [164].log_data[3].time := 3600.0, [164].log_data[3].valid := 1, [164].log_data[4].min := 0.64125, [164].log_data[4].max := 0.94875, [164].log_data[4].total := 3015.3088, [164].log_data[4].time := 3600.0, [164].log_data[4].maxminute := 59, [164].log_data[4].valid := 1, [164].log_data[5].max := 0.0012500001, [164].log_data[5].total := 0.22375216, [164].log_data[5].time := 3600.0, [164].log_data[5].valid := 1, [164].log_data[6].valid := 1, [164].log_data[7].valid := 1, [164].log_data[8].valid := 1, [164].log_data[9].valid := 1, [164].log_data[10].valid := 1, [164].log_data[11].valid := 1, [164].log_data[12].valid := 1, [164].log_data[13].valid := 1, [164].log_data[14].valid := 1,
        [164].log_data[15].valid := 1, [164].log_data[16].valid := 1, [164].log_data[17].valid := 1, [164].log_data[18].valid := 1, [164].log_data[19].valid := 1, [164].time.Year := 2022, [164].time.Month := 5, [164].time.Day := 3, [164].time.Hour := 13, [164].time.Minute := 59, [164].time.Second := 59, [164].time.DST_ON := 1, [165].log_data[0].min := 1.0, [165].log_data[0].max := 1.0, [165].log_data[0].total := 3600.0, [165].log_data[0].time := 3600.0, [165].log_data[0].valid := 1, [165].log_data[1].time := 3600.0, [165].log_data[1].valid := 1, [165].log_data[2].max := 1.0, [165].log_data[2].total := 477.0, [165].log_data[2].time := 3600.0, [165].log_data[2].maxminute := 35, [165].log_data[2].valid := 1, [165].log_data[3].time := 3600.0, [165].log_data[3].valid := 1, [165].log_data[4].min := 0.48749998, [165].log_data[4].max := 1.0068749, [165].log_data[4].total := 2975.2808, [165].log_data[4].time := 3600.0, [165].log_data[4].minminute := 43, [165].log_data[4].maxminute := 35, [165].log_data[4].valid := 1, [165].log_data[5].max := 7.275, [165].log_data[5].total := 3417.7673, [165].log_data[5].time := 3600.0, [165].log_data[5].maxminute := 37, [165].log_data[5].valid := 1, [165].log_data[6].valid := 1, [165].log_data[7].valid := 1, [165].log_data[8].valid := 1, [165].log_data[9].valid := 1, [165].log_data[10].valid := 1, [165].log_data[11].valid := 1, [165].log_data[12].valid := 1, [165].log_data[13].valid := 1, [165].log_data[14].valid := 1, [165].log_data[15].valid := 1, [165].log_data[16].valid := 1, [165].log_data[17].valid := 1, [165].log_data[18].valid := 1, [165].log_data[19].valid := 1, [165].time.Year := 2022, [165].time.Month := 5, [165].time.Day := 3, [165].time.Hour := 14, [165].time.Minute := 59, [165].time.Second := 59, [165].time.DST_ON := 1, [166].log_data[0].min := 1.0,
        [166].log_data[0].max := 1.0, [166].log_data[0].total := 3600.0, [166].log_data[0].time := 3600.0, [166].log_data[0].valid := 1, [166].log_data[1].time := 3600.0, [166].log_data[1].valid := 1, [166].log_data[2].time := 3600.0, [166].log_data[2].valid := 1, [166].log_data[3].time := 3600.0, [166].log_data[3].valid := 1, [166].log_data[4].min := 0.56437504, [166].log_data[4].max := 0.8725, [166].log_data[4].total := 2588.336, [166].log_data[4].time := 3600.0, [166].log_data[4].maxminute := 58, [166].log_data[4].valid := 1, [166].log_data[5].time := 3600.0, [166].log_data[5].valid := 1, [166].log_data[6].valid := 1, [166].log_data[7].valid := 1, [166].log_data[8].valid := 1, [166].log_data[9].valid := 1, [166].log_data[10].valid := 1, [166].log_data[11].valid := 1, [166].log_data[12].valid := 1, [166].log_data[13].valid := 1, [166].log_data[14].valid := 1, [166].log_data[15].valid := 1, [166].log_data[16].valid := 1, [166].log_data[17].valid := 1, [166].log_data[18].valid := 1, [166].log_data[19].valid := 1, [166].time.Year := 2022, [166].time.Month := 5, [166].time.Day := 3, [166].time.Hour := 15, [166].time.Minute := 59, [166].time.Second := 59, [166].time.DST_ON := 1, [167].log_data[0].min := 1.0, [167].log_data[0].max := 1.0, [167].log_data[0].total := 1798.5, [167].log_data[0].time := 1798.5, [167].log_data[0].valid := 1, [167].log_data[1].time := 1798.5, [167].log_data[1].valid := 1, [167].log_data[2].time := 1798.5, [167].log_data[2].valid := 1, [167].log_data[3].time := 1798.5, [167].log_data[3].valid := 1, [167].log_data[4].min := 0.871875, [167].log_data[4].max := 0.964375, [167].log_data[4].total := 1646.4832, [167].log_data[4].time := 1798.5, [167].log_data[4].maxminute := 29, [167].log_data[4].valid := 1, [167].log_data[5].time := 1798.5, [167].log_data[5].valid := 1, [167].log_data[6].valid := 1, [167].log_data[7].valid := 1,
        [167].log_data[8].valid := 1, [167].log_data[9].valid := 1, [167].log_data[10].valid := 1, [167].log_data[11].valid := 1, [167].log_data[12].valid := 1, [167].log_data[13].valid := 1, [167].log_data[14].valid := 1, [167].log_data[15].valid := 1, [167].log_data[16].valid := 1, [167].log_data[17].valid := 1, [167].log_data[18].valid := 1, [167].log_data[19].valid := 1, [168].log_data[0].min := 1.0, [168].log_data[0].max := 1.0, [168].log_data[0].total := 3600.001, [168].log_data[0].time := 3600.001, [168].log_data[0].valid := 1, [168].log_data[1].time := 3600.001, [168].log_data[1].valid := 1, [168].log_data[2].max := 1.0, [168].log_data[2].total := 495.0, [168].log_data[2].time := 3600.001, [168].log_data[2].maxminute := 28, [168].log_data[2].valid := 1, [168].log_data[3].time := 3600.001, [168].log_data[3].valid := 1, [168].log_data[4].min := 0.48749998, [168].log_data[4].max := 1.0081251, [168].log_data[4].total := 2849.0586, [168].log_data[4].time := 3600.001, [168].log_data[4].minminute := 36, [168].log_data[4].maxminute := 28, [168].log_data[4].valid := 1, [168].log_data[5].max := 7.2475, [168].log_data[5].total := 3526.0696, [168].log_data[5].time := 3600.001, [168].log_data[5].maxminute := 29, [168].log_data[5].valid := 1, [168].log_data[6].valid := 1, [168].log_data[7].valid := 1, [168].log_data[8].valid := 1, [168].log_data[9].valid := 1, [168].log_data[10].valid := 1, [168].log_data[11].valid := 1, [168].log_data[12].valid := 1, [168].log_data[13].valid := 1, [168].log_data[14].valid := 1, [168].log_data[15].valid := 1, [168].log_data[16].valid := 1, [168].log_data[17].valid := 1, [168].log_data[18].valid := 1, [168].log_data[19].valid := 1, [168].time.Year := 2022, [168].time.Month := 4, [168].time.Day := 25, [168].time.Hour := 9, [168].time.Minute := 59, [168].time.Second := 59, [168].time.DST_ON := 1, [169].log_data[0].min := 1.0,
        [169].log_data[0].max := 1.0, [169].log_data[0].total := 3600.0, [169].log_data[0].time := 3600.0, [169].log_data[0].valid := 1, [169].log_data[1].max := 1.0, [169].log_data[1].total := 500.5, [169].log_data[1].time := 3600.0, [169].log_data[1].maxminute := 43, [169].log_data[1].valid := 1, [169].log_data[2].time := 3600.0, [169].log_data[2].valid := 1, [169].log_data[3].time := 3600.0, [169].log_data[3].valid := 1, [169].log_data[4].min := 0.48687503, [169].log_data[4].max := 1.0081251, [169].log_data[4].total := 2981.0508, [169].log_data[4].time := 3600.0, [169].log_data[4].minminute := 53, [169].log_data[4].maxminute := 43, [169].log_data[4].valid := 1, [169].log_data[5].max := 7.2299995, [169].log_data[5].total := 3567.1848, [169].log_data[5].time := 3600.0, [169].log_data[5].maxminute := 44, [169].log_data[5].valid := 1, [169].log_data[6].valid := 1, [169].log_data[7].valid := 1, [169].log_data[8].valid := 1, [169].log_data[9].valid := 1, [169].log_data[10].valid := 1, [169].log_data[11].valid := 1, [169].log_data[12].valid := 1, [169].log_data[13].valid := 1, [169].log_data[14].valid := 1, [169].log_data[15].valid := 1, [169].log_data[16].valid := 1, [169].log_data[17].valid := 1, [169].log_data[18].valid := 1, [169].log_data[19].valid := 1, [169].time.Year := 2022, [169].time.Month := 4, [169].time.Day := 25, [169].time.Hour := 10, [169].time.Minute := 59, [169].time.Second := 59, [169].time.DST_ON := 1, [170].log_data[0].min := 1.0, [170].log_data[0].max := 1.0, [170].log_data[0].total := 3600.0, [170].log_data[0].time := 3600.0, [170].log_data[0].valid := 1, [170].log_data[1].time := 3600.0, [170].log_data[1].valid := 1, [170].log_data[2].time := 3600.0, [170].log_data[2].valid := 1, [170].log_data[3].time := 3600.0, [170].log_data[3].valid := 1, [170].log_data[4].min := 0.56437504, [170].log_data[4].max := 0.9637501, [170].log_data[4].total := 2878.8606,
        [170].log_data[4].time := 3600.0, [170].log_data[4].maxminute := 58, [170].log_data[4].valid := 1, [170].log_data[5].time := 3600.0, [170].log_data[5].valid := 1, [170].log_data[6].valid := 1, [170].log_data[7].valid := 1, [170].log_data[8].valid := 1, [170].log_data[9].valid := 1, [170].log_data[10].valid := 1, [170].log_data[11].valid := 1, [170].log_data[12].valid := 1, [170].log_data[13].valid := 1, [170].log_data[14].valid := 1, [170].log_data[15].valid := 1, [170].log_data[16].valid := 1, [170].log_data[17].valid := 1, [170].log_data[18].valid := 1, [170].log_data[19].valid := 1, [170].time.Year := 2022, [170].time.Month := 4, [170].time.Day := 25, [170].time.Hour := 11, [170].time.Minute := 59, [170].time.Second := 59, [170].time.DST_ON := 1, [171].log_data[0].min := 1.0, [171].log_data[0].max := 1.0, [171].log_data[0].total := 3600.0, [171].log_data[0].time := 3600.0, [171].log_data[0].valid := 1, [171].log_data[1].time := 3600.0, [171].log_data[1].valid := 1, [171].log_data[2].max := 1.0, [171].log_data[2].total := 492.0, [171].log_data[2].time := 3600.0, [171].log_data[2].maxminute := 10, [171].log_data[2].valid := 1, [171].log_data[3].time := 3600.0, [171].log_data[3].valid := 1, [171].log_data[4].min := 0.48687503, [171].log_data[4].max := 1.0068749, [171].log_data[4].total := 2552.135, [171].log_data[4].time := 3600.0, [171].log_data[4].minminute := 19, [171].log_data[4].maxminute := 10, [171].log_data[4].valid := 1, [171].log_data[5].max := 7.21875, [171].log_data[5].total := 3496.2583, [171].log_data[5].time := 3600.0, [171].log_data[5].maxminute := 11, [171].log_data[5].valid := 1, [171].log_data[6].valid := 1, [171].log_data[7].valid := 1, [171].log_data[8].valid := 1, [171].log_data[9].valid := 1, [171].log_data[10].valid := 1, [171].log_data[11].valid := 1, [171].log_data[12].valid := 1, [171].log_data[13].valid := 1,
        [171].log_data[14].valid := 1, [171].log_data[15].valid := 1, [171].log_data[16].valid := 1, [171].log_data[17].valid := 1, [171].log_data[18].valid := 1, [171].log_data[19].valid := 1, [171].time.Year := 2022, [171].time.Month := 4, [171].time.Day := 25, [171].time.Hour := 12, [171].time.Minute := 59, [171].time.Second := 59, [171].time.DST_ON := 1, [172].log_data[0].min := 1.0, [172].log_data[0].max := 1.0, [172].log_data[0].total := 3600.0, [172].log_data[0].time := 3600.0, [172].log_data[0].valid := 1, [172].log_data[1].time := 3600.0, [172].log_data[1].valid := 1, [172].log_data[2].time := 3600.0, [172].log_data[2].valid := 1, [172].log_data[3].time := 3600.0, [172].log_data[3].valid := 1, [172].log_data[4].min := 0.76375, [172].log_data[4].max := 0.97875005, [172].log_data[4].total := 3236.608, [172].log_data[4].time := 3600.0, [172].log_data[4].maxminute := 57, [172].log_data[4].valid := 1, [172].log_data[5].time := 3600.0, [172].log_data[5].valid := 1, [172].log_data[6].valid := 1, [172].log_data[7].valid := 1, [172].log_data[8].valid := 1, [172].log_data[9].valid := 1, [172].log_data[10].valid := 1, [172].log_data[11].valid := 1, [172].log_data[12].valid := 1, [172].log_data[13].valid := 1, [172].log_data[14].valid := 1, [172].log_data[15].valid := 1, [172].log_data[16].valid := 1, [172].log_data[17].valid := 1, [172].log_data[18].valid := 1, [172].log_data[19].valid := 1, [172].time.Year := 2022, [172].time.Month := 4, [172].time.Day := 25, [172].time.Hour := 13, [172].time.Minute := 59, [172].time.Second := 59, [172].time.DST_ON := 1, [173].log_data[0].min := 1.0, [173].log_data[0].max := 1.0, [173].log_data[0].total := 3599.999, [173].log_data[0].time := 3599.999, [173].log_data[0].valid := 1, [173].log_data[1].max := 1.0, [173].log_data[1].total := 486.0,
        [173].log_data[1].time := 3599.999, [173].log_data[1].maxminute := 14, [173].log_data[1].valid := 1, [173].log_data[2].time := 3599.999, [173].log_data[2].valid := 1, [173].log_data[3].time := 3599.999, [173].log_data[3].valid := 1, [173].log_data[4].min := 0.48687503, [173].log_data[4].max := 1.0081251, [173].log_data[4].total := 2547.991, [173].log_data[4].time := 3599.999, [173].log_data[4].minminute := 22, [173].log_data[4].maxminute := 14, [173].log_data[4].valid := 1, [173].log_data[5].max := 7.133749, [173].log_data[5].total := 3410.5862, [173].log_data[5].time := 3599.999, [173].log_data[5].maxminute := 15, [173].log_data[5].valid := 1, [173].log_data[6].valid := 1, [173].log_data[7].valid := 1, [173].log_data[8].valid := 1, [173].log_data[9].valid := 1, [173].log_data[10].valid := 1, [173].log_data[11].valid := 1, [173].log_data[12].valid := 1, [173].log_data[13].valid := 1, [173].log_data[14].valid := 1, [173].log_data[15].valid := 1, [173].log_data[16].valid := 1, [173].log_data[17].valid := 1, [173].log_data[18].valid := 1, [173].log_data[19].valid := 1, [173].time.Year := 2022, [173].time.Month := 4, [173].time.Day := 25, [173].time.Hour := 14, [173].time.Minute := 59, [173].time.Second := 59, [173].time.DST_ON := 1, [174].log_data[0].min := 1.0, [174].log_data[0].max := 1.0, [174].log_data[0].total := 3600.0, [174].log_data[0].time := 3600.0, [174].log_data[0].valid := 1, [174].log_data[1].time := 3600.0, [174].log_data[1].valid := 1, [174].log_data[2].time := 3600.0, [174].log_data[2].valid := 1, [174].log_data[3].time := 3600.0, [174].log_data[3].valid := 1, [174].log_data[4].min := 0.686875, [174].log_data[4].max := 0.918125, [174].log_data[4].total := 2958.2554, [174].log_data[4].time := 3600.0, [174].log_data[4].maxminute := 55, [174].log_data[4].valid := 1, [174].log_data[5].time := 3600.0, [174].log_data[5].valid := 1, [174].log_data[6].valid := 1,
        [174].log_data[7].valid := 1, [174].log_data[8].valid := 1, [174].log_data[9].valid := 1, [174].log_data[10].valid := 1, [174].log_data[11].valid := 1, [174].log_data[12].valid := 1, [174].log_data[13].valid := 1, [174].log_data[14].valid := 1, [174].log_data[15].valid := 1, [174].log_data[16].valid := 1, [174].log_data[17].valid := 1, [174].log_data[18].valid := 1, [174].log_data[19].valid := 1, [174].time.Year := 2022, [174].time.Month := 4, [174].time.Day := 25, [174].time.Hour := 15, [174].time.Minute := 59, [174].time.Second := 59, [174].time.DST_ON := 1, [175].log_data[0].min := 1.0, [175].log_data[0].max := 1.0, [175].log_data[0].total := 3600.0, [175].log_data[0].time := 3600.0, [175].log_data[0].valid := 1, [175].log_data[1].time := 3600.0, [175].log_data[1].valid := 1, [175].log_data[2].max := 1.0, [175].log_data[2].total := 494.5, [175].log_data[2].time := 3600.0, [175].log_data[2].maxminute := 37, [175].log_data[2].valid := 1, [175].log_data[3].time := 3600.0, [175].log_data[3].valid := 1, [175].log_data[4].min := 0.48687503, [175].log_data[4].max := 1.0081251, [175].log_data[4].total := 3032.2192, [175].log_data[4].time := 3600.0, [175].log_data[4].minminute := 45, [175].log_data[4].maxminute := 37, [175].log_data[4].valid := 1, [175].log_data[5].max := 7.30875, [175].log_data[5].total := 3559.0217, [175].log_data[5].time := 3600.0, [175].log_data[5].maxminute := 38, [175].log_data[5].valid := 1, [175].log_data[6].valid := 1, [175].log_data[7].valid := 1, [175].log_data[8].valid := 1, [175].log_data[9].valid := 1, [175].log_data[10].valid := 1, [175].log_data[11].valid := 1, [175].log_data[12].valid := 1, [175].log_data[13].valid := 1, [175].log_data[14].valid := 1, [175].log_data[15].valid := 1, [175].log_data[16].valid := 1, [175].log_data[17].valid := 1, [175].log_data[18].valid := 1, [175].log_data[19].valid := 1,
        [175].time.Year := 2022, [175].time.Month := 4, [175].time.Day := 25, [175].time.Hour := 16, [175].time.Minute := 59, [175].time.Second := 59, [175].time.DST_ON := 1, [176].log_data[0].min := 1.0, [176].log_data[0].max := 1.0, [176].log_data[0].total := 3600.0, [176].log_data[0].time := 3600.0, [176].log_data[0].valid := 1, [176].log_data[1].time := 3600.0, [176].log_data[1].valid := 1, [176].log_data[2].time := 3600.0, [176].log_data[2].valid := 1, [176].log_data[3].time := 3600.0, [176].log_data[3].valid := 1, [176].log_data[4].min := 0.625, [176].log_data[4].max := 0.97875005, [176].log_data[4].total := 3064.7, [176].log_data[4].time := 3600.0, [176].log_data[4].maxminute := 56, [176].log_data[4].valid := 1, [176].log_data[5].time := 3600.0, [176].log_data[5].valid := 1, [176].log_data[6].valid := 1, [176].log_data[7].valid := 1, [176].log_data[8].valid := 1, [176].log_data[9].valid := 1, [176].log_data[10].valid := 1, [176].log_data[11].valid := 1, [176].log_data[12].valid := 1, [176].log_data[13].valid := 1, [176].log_data[14].valid := 1, [176].log_data[15].valid := 1, [176].log_data[16].valid := 1, [176].log_data[17].valid := 1, [176].log_data[18].valid := 1, [176].log_data[19].valid := 1, [176].time.Year := 2022, [176].time.Month := 4, [176].time.Day := 25, [176].time.Hour := 17, [176].time.Minute := 59, [176].time.Second := 59, [176].time.DST_ON := 1, [177].log_data[0].min := 1.0, [177].log_data[0].max := 1.0, [177].log_data[0].total := 3600.0, [177].log_data[0].time := 3600.0, [177].log_data[0].valid := 1, [177].log_data[1].max := 1.0, [177].log_data[1].total := 490.5, [177].log_data[1].time := 3600.0, [177].log_data[1].maxminute := 8, [177].log_data[1].valid := 1, [177].log_data[2].time := 3600.0, [177].log_data[2].valid := 1, [177].log_data[3].time := 3600.0,
        [177].log_data[3].valid := 1, [177].log_data[4].min := 0.48687503, [177].log_data[4].max := 1.000625, [177].log_data[4].total := 2547.2048, [177].log_data[4].time := 3600.0, [177].log_data[4].minminute := 17, [177].log_data[4].maxminute := 8, [177].log_data[4].valid := 1, [177].log_data[5].max := 7.1237493, [177].log_data[5].total := 3436.7742, [177].log_data[5].time := 3600.0, [177].log_data[5].maxminute := 10, [177].log_data[5].valid := 1, [177].log_data[6].valid := 1, [177].log_data[7].valid := 1, [177].log_data[8].valid := 1, [177].log_data[9].valid := 1, [177].log_data[10].valid := 1, [177].log_data[11].valid := 1, [177].log_data[12].valid := 1, [177].log_data[13].valid := 1, [177].log_data[14].valid := 1, [177].log_data[15].valid := 1, [177].log_data[16].valid := 1, [177].log_data[17].valid := 1, [177].log_data[18].valid := 1, [177].log_data[19].valid := 1, [177].time.Year := 2022, [177].time.Month := 4, [177].time.Day := 25, [177].time.Hour := 18, [177].time.Minute := 59, [177].time.Second := 59, [177].time.DST_ON := 1, [178].log_data[0].min := 1.0, [178].log_data[0].max := 1.0, [178].log_data[0].total := 3600.0, [178].log_data[0].time := 3600.0, [178].log_data[0].valid := 1, [178].log_data[1].time := 3600.0, [178].log_data[1].valid := 1, [178].log_data[2].max := 1.0, [178].log_data[2].total := 503.0, [178].log_data[2].time := 3600.0, [178].log_data[2].maxminute := 40, [178].log_data[2].valid := 1, [178].log_data[3].time := 3600.0, [178].log_data[3].valid := 1, [178].log_data[4].min := 0.48687503, [178].log_data[4].max := 1.00625, [178].log_data[4].total := 2956.6802, [178].log_data[4].time := 3600.0, [178].log_data[4].minminute := 48, [178].log_data[4].maxminute := 40, [178].log_data[4].valid := 1, [178].log_data[5].max := 7.2087502, [178].log_data[5].total := 3567.3804, [178].log_data[5].time := 3600.0, [178].log_data[5].maxminute := 41, [178].log_data[5].valid := 1,
        [178].log_data[6].valid := 1, [178].log_data[7].valid := 1, [178].log_data[8].valid := 1, [178].log_data[9].valid := 1, [178].log_data[10].valid := 1, [178].log_data[11].valid := 1, [178].log_data[12].valid := 1, [178].log_data[13].valid := 1, [178].log_data[14].valid := 1, [178].log_data[15].valid := 1, [178].log_data[16].valid := 1, [178].log_data[17].valid := 1, [178].log_data[18].valid := 1, [178].log_data[19].valid := 1, [178].time.Year := 2022, [178].time.Month := 4, [178].time.Day := 25, [178].time.Hour := 19, [178].time.Minute := 59, [178].time.Second := 59, [178].time.DST_ON := 1, [179].log_data[0].min := 1.0, [179].log_data[0].max := 1.0, [179].log_data[0].total := 3600.0, [179].log_data[0].time := 3600.0, [179].log_data[0].valid := 1, [179].log_data[1].max := 1.0, [179].log_data[1].total := 524.5, [179].log_data[1].time := 3600.0, [179].log_data[1].maxminute := 44, [179].log_data[1].valid := 1, [179].log_data[2].time := 3600.0, [179].log_data[2].valid := 1, [179].log_data[3].time := 3600.0, [179].log_data[3].valid := 1, [179].log_data[4].min := 0.48749998, [179].log_data[4].max := 1.0081251, [179].log_data[4].total := 2773.5383, [179].log_data[4].time := 3600.0, [179].log_data[4].minminute := 53, [179].log_data[4].maxminute := 44, [179].log_data[4].valid := 1, [179].log_data[5].max := 7.1350007, [179].log_data[5].total := 3679.3784, [179].log_data[5].time := 3600.0, [179].log_data[5].maxminute := 45, [179].log_data[5].valid := 1, [179].log_data[6].valid := 1, [179].log_data[7].valid := 1, [179].log_data[8].valid := 1, [179].log_data[9].valid := 1, [179].log_data[10].valid := 1, [179].log_data[11].valid := 1, [179].log_data[12].valid := 1, [179].log_data[13].valid := 1, [179].log_data[14].valid := 1, [179].log_data[15].valid := 1, [179].log_data[16].valid := 1, [179].log_data[17].valid := 1, [179].log_data[18].valid := 1,
        [179].log_data[19].valid := 1, [179].time.Year := 2022, [179].time.Month := 4, [179].time.Day := 25, [179].time.Hour := 20, [179].time.Minute := 59, [179].time.Second := 59, [179].time.DST_ON := 1, [180].log_data[0].min := 1.0, [180].log_data[0].max := 1.0, [180].log_data[0].total := 3600.0, [180].log_data[0].time := 3600.0, [180].log_data[0].valid := 1, [180].log_data[1].time := 3600.0, [180].log_data[1].valid := 1, [180].log_data[2].max := 1.0, [180].log_data[2].total := 497.5, [180].log_data[2].time := 3600.0, [180].log_data[2].maxminute := 51, [180].log_data[2].valid := 1, [180].log_data[3].time := 3600.0, [180].log_data[3].valid := 1, [180].log_data[4].min := 0.48749998, [180].log_data[4].max := 1.0074999, [180].log_data[4].total := 2983.8057, [180].log_data[4].time := 3600.0, [180].log_data[4].minminute := 59, [180].log_data[4].maxminute := 51, [180].log_data[4].valid := 1, [180].log_data[5].max := 7.31375, [180].log_data[5].total := 3577.3186, [180].log_data[5].time := 3600.0, [180].log_data[5].maxminute := 52, [180].log_data[5].valid := 1, [180].log_data[6].valid := 1, [180].log_data[7].valid := 1, [180].log_data[8].valid := 1, [180].log_data[9].valid := 1, [180].log_data[10].valid := 1, [180].log_data[11].valid := 1, [180].log_data[12].valid := 1, [180].log_data[13].valid := 1, [180].log_data[14].valid := 1, [180].log_data[15].valid := 1, [180].log_data[16].valid := 1, [180].log_data[17].valid := 1, [180].log_data[18].valid := 1, [180].log_data[19].valid := 1, [180].time.Year := 2022, [180].time.Month := 4, [180].time.Day := 25, [180].time.Hour := 21, [180].time.Minute := 59, [180].time.Second := 59, [180].time.DST_ON := 1, [181].log_data[0].min := 1.0, [181].log_data[0].max := 1.0, [181].log_data[0].total := 3600.0, [181].log_data[0].time := 3600.0, [181].log_data[0].valid := 1,
        [181].log_data[1].time := 3600.0, [181].log_data[1].valid := 1, [181].log_data[2].time := 3600.0, [181].log_data[2].valid := 1, [181].log_data[3].time := 3600.0, [181].log_data[3].valid := 1, [181].log_data[4].min := 0.48749998, [181].log_data[4].max := 0.97937495, [181].log_data[4].total := 2736.6736, [181].log_data[4].time := 3600.0, [181].log_data[4].maxminute := 59, [181].log_data[4].valid := 1, [181].log_data[5].max := 0.0012500001, [181].log_data[5].total := 0.0028125, [181].log_data[5].time := 3600.0, [181].log_data[5].maxminute := 16, [181].log_data[5].valid := 1, [181].log_data[6].valid := 1, [181].log_data[7].valid := 1, [181].log_data[8].valid := 1, [181].log_data[9].valid := 1, [181].log_data[10].valid := 1, [181].log_data[11].valid := 1, [181].log_data[12].valid := 1, [181].log_data[13].valid := 1, [181].log_data[14].valid := 1, [181].log_data[15].valid := 1, [181].log_data[16].valid := 1, [181].log_data[17].valid := 1, [181].log_data[18].valid := 1, [181].log_data[19].valid := 1, [181].time.Year := 2022, [181].time.Month := 4, [181].time.Day := 25, [181].time.Hour := 22, [181].time.Minute := 59, [181].time.Second := 59, [181].time.DST_ON := 1, [182].log_data[0].min := 1.0, [182].log_data[0].max := 1.0, [182].log_data[0].total := 3600.0, [182].log_data[0].time := 3600.0, [182].log_data[0].valid := 1, [182].log_data[1].max := 1.0, [182].log_data[1].total := 509.0, [182].log_data[1].time := 3600.0, [182].log_data[1].maxminute := 6, [182].log_data[1].valid := 1, [182].log_data[2].time := 3600.0, [182].log_data[2].valid := 1, [182].log_data[3].time := 3600.0, [182].log_data[3].valid := 1, [182].log_data[4].min := 0.48749998, [182].log_data[4].max := 1.00875, [182].log_data[4].total := 2647.123, [182].log_data[4].time := 3600.0, [182].log_data[4].minminute := 15, [182].log_data[4].maxminute := 6, [182].log_data[4].valid := 1, [182].log_data[5].max := 7.1350007,
        [182].log_data[5].total := 3571.7212, [182].log_data[5].time := 3600.0, [182].log_data[5].maxminute := 7, [182].log_data[5].valid := 1, [182].log_data[6].valid := 1, [182].log_data[7].valid := 1, [182].log_data[8].valid := 1, [182].log_data[9].valid := 1, [182].log_data[10].valid := 1, [182].log_data[11].valid := 1, [182].log_data[12].valid := 1, [182].log_data[13].valid := 1, [182].log_data[14].valid := 1, [182].log_data[15].valid := 1, [182].log_data[16].valid := 1, [182].log_data[17].valid := 1, [182].log_data[18].valid := 1, [182].log_data[19].valid := 1, [182].time.Year := 2022, [182].time.Month := 4, [182].time.Day := 25, [182].time.Hour := 23, [182].time.Minute := 59, [182].time.Second := 59, [182].time.DST_ON := 1, [183].log_data[0].min := 1.0, [183].log_data[0].max := 1.0, [183].log_data[0].total := 3599.999, [183].log_data[0].time := 3599.999, [183].log_data[0].valid := 1, [183].log_data[1].time := 3599.999, [183].log_data[1].valid := 1, [183].log_data[2].max := 1.0, [183].log_data[2].total := 58.25, [183].log_data[2].time := 3599.999, [183].log_data[2].maxminute := 59, [183].log_data[2].valid := 1, [183].log_data[3].time := 3599.999, [183].log_data[3].valid := 1, [183].log_data[4].min := 0.85625, [183].log_data[4].max := 1.0068749, [183].log_data[4].total := 3372.4036, [183].log_data[4].time := 3599.999, [183].log_data[4].maxminute := 59, [183].log_data[4].valid := 1, [183].log_data[5].max := 7.20125, [183].log_data[5].total := 357.3134, [183].log_data[5].time := 3599.999, [183].log_data[5].maxminute := 59, [183].log_data[5].valid := 1, [183].log_data[6].valid := 1, [183].log_data[7].valid := 1, [183].log_data[8].valid := 1, [183].log_data[9].valid := 1, [183].log_data[10].valid := 1, [183].log_data[11].valid := 1, [183].log_data[12].valid := 1, [183].log_data[13].valid := 1, [183].log_data[14].valid := 1, [183].log_data[15].valid := 1,
        [183].log_data[16].valid := 1, [183].log_data[17].valid := 1, [183].log_data[18].valid := 1, [183].log_data[19].valid := 1, [183].time.Year := 2022, [183].time.Month := 4, [183].time.Day := 26, [183].time.Minute := 59, [183].time.Second := 59, [183].time.DST_ON := 1, [184].log_data[0].min := 1.0, [184].log_data[0].max := 1.0, [184].log_data[0].total := 3600.0, [184].log_data[0].time := 3600.0, [184].log_data[0].valid := 1, [184].log_data[1].time := 3600.0, [184].log_data[1].valid := 1, [184].log_data[2].max := 1.0, [184].log_data[2].total := 422.75, [184].log_data[2].time := 3600.0, [184].log_data[2].minminute := 7, [184].log_data[2].valid := 1, [184].log_data[3].time := 3600.0, [184].log_data[3].valid := 1, [184].log_data[4].min := 0.479375, [184].log_data[4].max := 0.9668751, [184].log_data[4].total := 2358.224, [184].log_data[4].time := 3600.0, [184].log_data[4].minminute := 7, [184].log_data[4].valid := 1, [184].log_data[5].max := 7.2087502, [184].log_data[5].total := 3060.4253, [184].log_data[5].time := 3600.0, [184].log_data[5].minminute := 7, [184].log_data[5].valid := 1, [184].log_data[6].valid := 1, [184].log_data[7].valid := 1, [184].log_data[8].valid := 1, [184].log_data[9].valid := 1, [184].log_data[10].valid := 1, [184].log_data[11].valid := 1, [184].log_data[12].valid := 1, [184].log_data[13].valid := 1, [184].log_data[14].valid := 1, [184].log_data[15].valid := 1, [184].log_data[16].valid := 1, [184].log_data[17].valid := 1, [184].log_data[18].valid := 1, [184].log_data[19].valid := 1, [184].time.Year := 2022, [184].time.Month := 4, [184].time.Day := 26, [184].time.Hour := 1, [184].time.Minute := 59, [184].time.Second := 59, [184].time.DST_ON := 1, [185].log_data[0].min := 1.0, [185].log_data[0].max := 1.0, [185].log_data[0].total := 3600.001, [185].log_data[0].time := 3600.001,
        [185].log_data[0].valid := 1, [185].log_data[1].time := 3600.001, [185].log_data[1].valid := 1, [185].log_data[2].time := 3600.001, [185].log_data[2].valid := 1, [185].log_data[3].time := 3600.001, [185].log_data[3].valid := 1, [185].log_data[4].min := 0.79499996, [185].log_data[4].max := 0.964375, [185].log_data[4].total := 3237.4219, [185].log_data[4].time := 3600.001, [185].log_data[4].maxminute := 58, [185].log_data[4].valid := 1, [185].log_data[5].max := 0.0012500001, [185].log_data[5].total := 0.2568779, [185].log_data[5].time := 3600.001, [185].log_data[5].valid := 1, [185].log_data[6].valid := 1, [185].log_data[7].valid := 1, [185].log_data[8].valid := 1, [185].log_data[9].valid := 1, [185].log_data[10].valid := 1, [185].log_data[11].valid := 1, [185].log_data[12].valid := 1, [185].log_data[13].valid := 1, [185].log_data[14].valid := 1, [185].log_data[15].valid := 1, [185].log_data[16].valid := 1, [185].log_data[17].valid := 1, [185].log_data[18].valid := 1, [185].log_data[19].valid := 1, [185].time.Year := 2022, [185].time.Month := 4, [185].time.Day := 26, [185].time.Hour := 2, [185].time.Minute := 59, [185].time.Second := 59, [185].time.DST_ON := 1, [186].log_data[0].min := 1.0, [186].log_data[0].max := 1.0, [186].log_data[0].total := 3600.0, [186].log_data[0].time := 3600.0, [186].log_data[0].valid := 1, [186].log_data[1].max := 1.0, [186].log_data[1].total := 477.0, [186].log_data[1].time := 3600.0, [186].log_data[1].maxminute := 35, [186].log_data[1].valid := 1, [186].log_data[2].time := 3600.0, [186].log_data[2].valid := 1, [186].log_data[3].time := 3600.0, [186].log_data[3].valid := 1, [186].log_data[4].min := 0.48749998, [186].log_data[4].max := 1.005, [186].log_data[4].total := 2966.531, [186].log_data[4].time := 3600.0, [186].log_data[4].minminute := 43, [186].log_data[4].maxminute := 35, [186].log_data[4].valid := 1, [186].log_data[5].max := 7.1425004,
        [186].log_data[5].total := 3353.21, [186].log_data[5].time := 3600.0, [186].log_data[5].maxminute := 35, [186].log_data[5].valid := 1, [186].log_data[6].valid := 1, [186].log_data[7].valid := 1, [186].log_data[8].valid := 1, [186].log_data[9].valid := 1, [186].log_data[10].valid := 1, [186].log_data[11].valid := 1, [186].log_data[12].valid := 1, [186].log_data[13].valid := 1, [186].log_data[14].valid := 1, [186].log_data[15].valid := 1, [186].log_data[16].valid := 1, [186].log_data[17].valid := 1, [186].log_data[18].valid := 1, [186].log_data[19].valid := 1, [186].time.Year := 2022, [186].time.Month := 4, [186].time.Day := 26, [186].time.Hour := 3, [186].time.Minute := 59, [186].time.Second := 59, [186].time.DST_ON := 1, [187].log_data[0].min := 1.0, [187].log_data[0].max := 1.0, [187].log_data[0].total := 3600.0, [187].log_data[0].time := 3600.0, [187].log_data[0].valid := 1, [187].log_data[1].time := 3600.0, [187].log_data[1].valid := 1, [187].log_data[2].time := 3600.0, [187].log_data[2].valid := 1, [187].log_data[3].time := 3600.0, [187].log_data[3].valid := 1, [187].log_data[4].min := 0.53374994, [187].log_data[4].max := 0.713125, [187].log_data[4].total := 2276.4612, [187].log_data[4].time := 3600.0, [187].log_data[4].maxminute := 59, [187].log_data[4].valid := 1, [187].log_data[5].max := 0.0012500001, [187].log_data[5].total := 0.059062455, [187].log_data[5].time := 3600.0, [187].log_data[5].valid := 1, [187].log_data[6].valid := 1, [187].log_data[7].valid := 1, [187].log_data[8].valid := 1, [187].log_data[9].valid := 1, [187].log_data[10].valid := 1, [187].log_data[11].valid := 1, [187].log_data[12].valid := 1, [187].log_data[13].valid := 1, [187].log_data[14].valid := 1, [187].log_data[15].valid := 1, [187].log_data[16].valid := 1, [187].log_data[17].valid := 1, [187].log_data[18].valid := 1, [187].log_data[19].valid := 1,
        [187].time.Year := 2022, [187].time.Month := 4, [187].time.Day := 26, [187].time.Hour := 4, [187].time.Minute := 59, [187].time.Second := 59, [187].time.DST_ON := 1, [188].log_data[0].min := 1.0, [188].log_data[0].max := 1.0, [188].log_data[0].total := 3600.0, [188].log_data[0].time := 3600.0, [188].log_data[0].valid := 1, [188].log_data[1].time := 3600.0, [188].log_data[1].valid := 1, [188].log_data[2].time := 3600.0, [188].log_data[2].valid := 1, [188].log_data[3].time := 3600.0, [188].log_data[3].valid := 1, [188].log_data[4].min := 0.713125, [188].log_data[4].max := 0.84124994, [188].log_data[4].total := 2791.2856, [188].log_data[4].time := 3600.0, [188].log_data[4].maxminute := 55, [188].log_data[4].valid := 1, [188].log_data[5].max := 0.0012500001, [188].log_data[5].total := 0.116562404, [188].log_data[5].time := 3600.0, [188].log_data[5].valid := 1, [188].log_data[6].valid := 1, [188].log_data[7].valid := 1, [188].log_data[8].valid := 1, [188].log_data[9].valid := 1, [188].log_data[10].valid := 1, [188].log_data[11].valid := 1, [188].log_data[12].valid := 1, [188].log_data[13].valid := 1, [188].log_data[14].valid := 1, [188].log_data[15].valid := 1, [188].log_data[16].valid := 1, [188].log_data[17].valid := 1, [188].log_data[18].valid := 1, [188].log_data[19].valid := 1, [188].time.Year := 2022, [188].time.Month := 4, [188].time.Day := 26, [188].time.Hour := 5, [188].time.Minute := 59, [188].time.Second := 59, [188].time.DST_ON := 1, [189].log_data[0].min := 1.0, [189].log_data[0].max := 1.0, [189].log_data[0].total := 3600.0, [189].log_data[0].time := 3600.0, [189].log_data[0].valid := 1, [189].log_data[1].time := 3600.0, [189].log_data[1].valid := 1, [189].log_data[2].time := 3600.0, [189].log_data[2].valid := 1, [189].log_data[3].time := 3600.0, [189].log_data[3].valid := 1,
        [189].log_data[4].min := 0.84062505, [189].log_data[4].max := 0.93375, [189].log_data[4].total := 3239.4949, [189].log_data[4].time := 3600.0, [189].log_data[4].maxminute := 49, [189].log_data[4].valid := 1, [189].log_data[5].max := 0.0012500001, [189].log_data[5].total := 0.13781269, [189].log_data[5].time := 3600.0, [189].log_data[5].valid := 1, [189].log_data[6].valid := 1, [189].log_data[7].valid := 1, [189].log_data[8].valid := 1, [189].log_data[9].valid := 1, [189].log_data[10].valid := 1, [189].log_data[11].valid := 1, [189].log_data[12].valid := 1, [189].log_data[13].valid := 1, [189].log_data[14].valid := 1, [189].log_data[15].valid := 1, [189].log_data[16].valid := 1, [189].log_data[17].valid := 1, [189].log_data[18].valid := 1, [189].log_data[19].valid := 1, [189].time.Year := 2022, [189].time.Month := 4, [189].time.Day := 26, [189].time.Hour := 6, [189].time.Minute := 59, [189].time.Second := 59, [189].time.DST_ON := 1, [190].log_data[0].min := 1.0, [190].log_data[0].max := 1.0, [190].log_data[0].total := 3600.0, [190].log_data[0].time := 3600.0, [190].log_data[0].valid := 1, [190].log_data[1].time := 3600.0, [190].log_data[1].valid := 1, [190].log_data[2].max := 1.0, [190].log_data[2].total := 82.25, [190].log_data[2].time := 3600.0, [190].log_data[2].maxminute := 58, [190].log_data[2].valid := 1, [190].log_data[3].time := 3600.0, [190].log_data[3].valid := 1, [190].log_data[4].min := 0.933125, [190].log_data[4].max := 1.005, [190].log_data[4].total := 3488.375, [190].log_data[4].time := 3600.0, [190].log_data[4].maxminute := 58, [190].log_data[4].valid := 1, [190].log_data[5].max := 7.2275, [190].log_data[5].total := 531.06256, [190].log_data[5].time := 3600.0, [190].log_data[5].maxminute := 59, [190].log_data[5].valid := 1, [190].log_data[6].valid := 1, [190].log_data[7].valid := 1, [190].log_data[8].valid := 1, [190].log_data[9].valid := 1,
        [190].log_data[10].valid := 1, [190].log_data[11].valid := 1, [190].log_data[12].valid := 1, [190].log_data[13].valid := 1, [190].log_data[14].valid := 1, [190].log_data[15].valid := 1, [190].log_data[16].valid := 1, [190].log_data[17].valid := 1, [190].log_data[18].valid := 1, [190].log_data[19].valid := 1, [190].time.Year := 2022, [190].time.Month := 4, [190].time.Day := 26, [190].time.Hour := 7, [190].time.Minute := 59, [190].time.Second := 59, [190].time.DST_ON := 1, [191].log_data[0].min := 1.0, [191].log_data[0].max := 1.0, [191].log_data[0].total := 3600.0, [191].log_data[0].time := 3600.0, [191].log_data[0].valid := 1, [191].log_data[1].time := 3600.0, [191].log_data[1].valid := 1, [191].log_data[2].max := 1.0, [191].log_data[2].total := 395.75, [191].log_data[2].time := 3600.0, [191].log_data[2].minminute := 6, [191].log_data[2].valid := 1, [191].log_data[3].time := 3600.0, [191].log_data[3].valid := 1, [191].log_data[4].min := 0.48749998, [191].log_data[4].max := 0.964375, [191].log_data[4].total := 2406.61, [191].log_data[4].time := 3600.0, [191].log_data[4].minminute := 7, [191].log_data[4].valid := 1, [191].log_data[5].max := 7.2199993, [191].log_data[5].total := 2866.0215, [191].log_data[5].time := 3600.0, [191].log_data[5].minminute := 6, [191].log_data[5].valid := 1, [191].log_data[6].valid := 1, [191].log_data[7].valid := 1, [191].log_data[8].valid := 1, [191].log_data[9].valid := 1, [191].log_data[10].valid := 1, [191].log_data[11].valid := 1, [191].log_data[12].valid := 1, [191].log_data[13].valid := 1, [191].log_data[14].valid := 1, [191].log_data[15].valid := 1, [191].log_data[16].valid := 1, [191].log_data[17].valid := 1, [191].log_data[18].valid := 1, [191].log_data[19].valid := 1, [191].time.Year := 2022, [191].time.Month := 4, [191].time.Day := 26, [191].time.Hour := 8,
        [191].time.Minute := 59, [191].time.Second := 59, [191].time.DST_ON := 1, [192].log_data[0].min := 1.0, [192].log_data[0].max := 1.0, [192].log_data[0].total := 3600.0, [192].log_data[0].time := 3600.0, [192].log_data[0].valid := 1, [192].log_data[1].max := 1.0, [192].log_data[1].total := 506.0, [192].log_data[1].time := 3600.0, [192].log_data[1].maxminute := 23, [192].log_data[1].valid := 1, [192].log_data[2].time := 3600.0, [192].log_data[2].valid := 1, [192].log_data[3].time := 3600.0, [192].log_data[3].valid := 1, [192].log_data[4].min := 0.48749998, [192].log_data[4].max := 1.0068749, [192].log_data[4].total := 2758.246, [192].log_data[4].time := 3600.0, [192].log_data[4].minminute := 32, [192].log_data[4].maxminute := 23, [192].log_data[4].valid := 1, [192].log_data[5].max := 7.1375, [192].log_data[5].total := 3551.0176, [192].log_data[5].time := 3600.0, [192].log_data[5].maxminute := 24, [192].log_data[5].valid := 1, [192].log_data[6].valid := 1, [192].log_data[7].valid := 1, [192].log_data[8].valid := 1, [192].log_data[9].valid := 1, [192].log_data[10].valid := 1, [192].log_data[11].valid := 1, [192].log_data[12].valid := 1, [192].log_data[13].valid := 1, [192].log_data[14].valid := 1, [192].log_data[15].valid := 1, [192].log_data[16].valid := 1, [192].log_data[17].valid := 1, [192].log_data[18].valid := 1, [192].log_data[19].valid := 1, [192].time.Year := 2022, [192].time.Month := 4, [192].time.Day := 26, [192].time.Hour := 9, [192].time.Minute := 59, [192].time.Second := 59, [192].time.DST_ON := 1, [193].log_data[0].min := 1.0, [193].log_data[0].max := 1.0, [193].log_data[0].total := 3600.0, [193].log_data[0].time := 3600.0, [193].log_data[0].valid := 1, [193].log_data[1].time := 3600.0, [193].log_data[1].valid := 1, [193].log_data[2].max := 1.0, [193].log_data[2].total := 495.0, [193].log_data[2].time := 3600.0,
        [193].log_data[2].maxminute := 49, [193].log_data[2].valid := 1, [193].log_data[3].time := 3600.0, [193].log_data[3].valid := 1, [193].log_data[4].min := 0.48749998, [193].log_data[4].max := 1.0074999, [193].log_data[4].total := 3049.0813, [193].log_data[4].time := 3600.0, [193].log_data[4].minminute := 57, [193].log_data[4].maxminute := 49, [193].log_data[4].valid := 1, [193].log_data[5].max := 7.2225, [193].log_data[5].total := 3517.6877, [193].log_data[5].time := 3600.0, [193].log_data[5].maxminute := 52, [193].log_data[5].valid := 1, [193].log_data[6].valid := 1, [193].log_data[7].valid := 1, [193].log_data[8].valid := 1, [193].log_data[9].valid := 1, [193].log_data[10].valid := 1, [193].log_data[11].valid := 1, [193].log_data[12].valid := 1, [193].log_data[13].valid := 1, [193].log_data[14].valid := 1, [193].log_data[15].valid := 1, [193].log_data[16].valid := 1, [193].log_data[17].valid := 1, [193].log_data[18].valid := 1, [193].log_data[19].valid := 1, [193].time.Year := 2022, [193].time.Month := 4, [193].time.Day := 26, [193].time.Hour := 10, [193].time.Minute := 59, [193].time.Second := 59, [193].time.DST_ON := 1, [194].log_data[0].min := 1.0, [194].log_data[0].max := 1.0, [194].log_data[0].total := 3600.0, [194].log_data[0].time := 3600.0, [194].log_data[0].valid := 1, [194].log_data[1].max := 1.0, [194].log_data[1].total := 464.25, [194].log_data[1].time := 3600.0, [194].log_data[1].maxminute := 1, [194].log_data[1].valid := 1, [194].log_data[2].time := 3600.0, [194].log_data[2].valid := 1, [194].log_data[3].time := 3600.0, [194].log_data[3].valid := 1, [194].log_data[4].min := 0.0725, [194].log_data[4].max := 0.50374997, [194].log_data[4].total := 858.2045, [194].log_data[4].time := 3600.0, [194].log_data[4].minminute := 7, [194].log_data[4].valid := 1, [194].log_data[5].max := 6.942499, [194].log_data[5].total := 2226.2878, [194].log_data[5].time := 3600.0,
        [194].log_data[5].maxminute := 2, [194].log_data[5].valid := 1, [194].log_data[6].valid := 1, [194].log_data[7].valid := 1, [194].log_data[8].valid := 1, [194].log_data[9].valid := 1, [194].log_data[10].valid := 1, [194].log_data[11].valid := 1, [194].log_data[12].valid := 1, [194].log_data[13].valid := 1, [194].log_data[14].valid := 1, [194].log_data[15].valid := 1, [194].log_data[16].valid := 1, [194].log_data[17].valid := 1, [194].log_data[18].valid := 1, [194].log_data[19].valid := 1, [194].time.Year := 2022, [194].time.Month := 4, [194].time.Day := 26, [194].time.Hour := 11, [194].time.Minute := 59, [194].time.Second := 59, [194].time.DST_ON := 1, [195].log_data[0].min := 1.0, [195].log_data[0].max := 1.0, [195].log_data[0].total := 3600.0, [195].log_data[0].time := 3600.0, [195].log_data[0].valid := 1, [195].log_data[1].time := 3600.0, [195].log_data[1].valid := 1, [195].log_data[2].time := 3600.0, [195].log_data[2].valid := 1, [195].log_data[3].time := 3600.0, [195].log_data[3].valid := 1, [195].log_data[4].min := 0.395625, [195].log_data[4].max := 0.87125003, [195].log_data[4].total := 2335.6277, [195].log_data[4].time := 3600.0, [195].log_data[4].maxminute := 59, [195].log_data[4].valid := 1, [195].log_data[5].time := 3600.0, [195].log_data[5].valid := 1, [195].log_data[6].valid := 1, [195].log_data[7].valid := 1, [195].log_data[8].valid := 1, [195].log_data[9].valid := 1, [195].log_data[10].valid := 1, [195].log_data[11].valid := 1, [195].log_data[12].valid := 1, [195].log_data[13].valid := 1, [195].log_data[14].valid := 1, [195].log_data[15].valid := 1, [195].log_data[16].valid := 1, [195].log_data[17].valid := 1, [195].log_data[18].valid := 1, [195].log_data[19].valid := 1, [195].time.Year := 2022, [195].time.Month := 4, [195].time.Day := 26, [195].time.Hour := 12,
        [195].time.Minute := 59, [195].time.Second := 59, [195].time.DST_ON := 1, [196].log_data[0].min := 1.0, [196].log_data[0].max := 1.0, [196].log_data[0].total := 3600.0, [196].log_data[0].time := 3600.0, [196].log_data[0].valid := 1, [196].log_data[1].max := 1.0, [196].log_data[1].total := 480.5, [196].log_data[1].time := 3600.0, [196].log_data[1].maxminute := 41, [196].log_data[1].valid := 1, [196].log_data[2].time := 3600.0, [196].log_data[2].valid := 1, [196].log_data[3].time := 3600.0, [196].log_data[3].valid := 1, [196].log_data[4].min := 0.48749998, [196].log_data[4].max := 1.00625, [196].log_data[4].total := 3070.715, [196].log_data[4].time := 3600.0, [196].log_data[4].minminute := 50, [196].log_data[4].maxminute := 42, [196].log_data[4].valid := 1, [196].log_data[5].max := 7.2250004, [196].log_data[5].total := 3401.9412, [196].log_data[5].time := 3600.0, [196].log_data[5].maxminute := 43, [196].log_data[5].valid := 1, [196].log_data[6].valid := 1, [196].log_data[7].valid := 1, [196].log_data[8].valid := 1, [196].log_data[9].valid := 1, [196].log_data[10].valid := 1, [196].log_data[11].valid := 1, [196].log_data[12].valid := 1, [196].log_data[13].valid := 1, [196].log_data[14].valid := 1, [196].log_data[15].valid := 1, [196].log_data[16].valid := 1, [196].log_data[17].valid := 1, [196].log_data[18].valid := 1, [196].log_data[19].valid := 1, [196].time.Year := 2022, [196].time.Month := 4, [196].time.Day := 26, [196].time.Hour := 13, [196].time.Minute := 59, [196].time.Second := 59, [196].time.DST_ON := 1, [197].log_data[0].min := 1.0, [197].log_data[0].max := 1.0, [197].log_data[0].total := 3600.0, [197].log_data[0].time := 3600.0, [197].log_data[0].valid := 1, [197].log_data[1].time := 3600.0, [197].log_data[1].valid := 1, [197].log_data[2].time := 3600.0, [197].log_data[2].valid := 1, [197].log_data[3].time := 3600.0,
        [197].log_data[3].valid := 1, [197].log_data[4].min := 0.54812497, [197].log_data[4].max := 0.91875005, [197].log_data[4].total := 2660.6123, [197].log_data[4].time := 3600.0, [197].log_data[4].maxminute := 57, [197].log_data[4].valid := 1, [197].log_data[5].time := 3600.0, [197].log_data[5].valid := 1, [197].log_data[6].valid := 1, [197].log_data[7].valid := 1, [197].log_data[8].valid := 1, [197].log_data[9].valid := 1, [197].log_data[10].valid := 1, [197].log_data[11].valid := 1, [197].log_data[12].valid := 1, [197].log_data[13].valid := 1, [197].log_data[14].valid := 1, [197].log_data[15].valid := 1, [197].log_data[16].valid := 1, [197].log_data[17].valid := 1, [197].log_data[18].valid := 1, [197].log_data[19].valid := 1, [197].time.Year := 2022, [197].time.Month := 4, [197].time.Day := 26, [197].time.Hour := 14, [197].time.Minute := 59, [197].time.Second := 59, [197].time.DST_ON := 1, [198].log_data[0].min := 1.0, [198].log_data[0].max := 1.0, [198].log_data[0].total := 3600.0, [198].log_data[0].time := 3600.0, [198].log_data[0].valid := 1, [198].log_data[1].time := 3600.0, [198].log_data[1].valid := 1, [198].log_data[2].max := 1.0, [198].log_data[2].total := 481.0, [198].log_data[2].time := 3600.0, [198].log_data[2].maxminute := 37, [198].log_data[2].valid := 1, [198].log_data[3].time := 3600.0, [198].log_data[3].valid := 1, [198].log_data[4].min := 0.48749998, [198].log_data[4].max := 1.0068749, [198].log_data[4].total := 2999.3838, [198].log_data[4].time := 3600.0, [198].log_data[4].minminute := 45, [198].log_data[4].maxminute := 37, [198].log_data[4].valid := 1, [198].log_data[5].max := 7.2299995, [198].log_data[5].total := 3385.684, [198].log_data[5].time := 3600.0, [198].log_data[5].maxminute := 38, [198].log_data[5].valid := 1, [198].log_data[6].valid := 1, [198].log_data[7].valid := 1, [198].log_data[8].valid := 1, [198].log_data[9].valid := 1,
        [198].log_data[10].valid := 1, [198].log_data[11].valid := 1, [198].log_data[12].valid := 1, [198].log_data[13].valid := 1, [198].log_data[14].valid := 1, [198].log_data[15].valid := 1, [198].log_data[16].valid := 1, [198].log_data[17].valid := 1, [198].log_data[18].valid := 1, [198].log_data[19].valid := 1, [198].time.Year := 2022, [198].time.Month := 4, [198].time.Day := 26, [198].time.Hour := 15, [198].time.Minute := 59, [198].time.Second := 59, [198].time.DST_ON := 1, [199].log_data[0].min := 1.0, [199].log_data[0].max := 1.0, [199].log_data[0].total := 3600.0, [199].log_data[0].time := 3600.0, [199].log_data[0].valid := 1, [199].log_data[1].time := 3600.0, [199].log_data[1].valid := 1, [199].log_data[2].time := 3600.0, [199].log_data[2].valid := 1, [199].log_data[3].time := 3600.0, [199].log_data[3].valid := 1, [199].log_data[4].min := 0.56437504, [199].log_data[4].max := 0.8875, [199].log_data[4].total := 2583.2231, [199].log_data[4].time := 3600.0, [199].log_data[4].maxminute := 59, [199].log_data[4].valid := 1, [199].log_data[5].max := 0.0012500001, [199].log_data[5].total := 0.00062500004, [199].log_data[5].time := 3600.0, [199].log_data[5].maxminute := 32, [199].log_data[5].valid := 1, [199].log_data[6].valid := 1, [199].log_data[7].valid := 1, [199].log_data[8].valid := 1, [199].log_data[9].valid := 1, [199].log_data[10].valid := 1, [199].log_data[11].valid := 1, [199].log_data[12].valid := 1, [199].log_data[13].valid := 1, [199].log_data[14].valid := 1, [199].log_data[15].valid := 1, [199].log_data[16].valid := 1, [199].log_data[17].valid := 1, [199].log_data[18].valid := 1, [199].log_data[19].valid := 1, [199].time.Year := 2022, [199].time.Month := 4, [199].time.Day := 26, [199].time.Hour := 16, [199].time.Minute := 59, [199].time.Second := 59, [199].time.DST_ON := 1);
   report_pwrup_done : BOOL := 1;
   report_row_qty : DINT := 200;
   report_tag_qty : DINT := 20;
   sequence_pwrup_done : BOOL := 1;
   SoftwareFault : BOOL;   // System software fault
   TO_QW360 : COMMBLOCK := (WATCHDOG := 450, REALS[0] := 0.963125);
   valve_pwrup_done : BOOL := 1;
   WALLCLOCK : DateTime := (Year := 2022, Month := 5, Day := 3, Hour := 16, Minute := 29, Second := 57, Microsecond := 121912, DayOfWeek := 2, DST_ON := 1);   // Global date / time
   WALLCLOCK_lock : BOOL;
   Watchdog_Relay : BOOL;
   XAFLOAT : ALM := (enmn := 1, chan := 6, enau := 1, alarm_tonr.TimerEnable := 1, alarm_tonr.Reset := 1);   // Station in float mode
   XAHWARE : ALM := (raw := 1, enau := 1, alarm_tonr.TimerEnable := 1, alarm_tonr.Reset := 1);   // PLC hardware fault
   XASWARE : ALM := (enmn := 1, enau := 1, alarm_tonr.TimerEnable := 1, alarm_tonr.Reset := 1);   // PLC software fault
END_VAR
